LIN {X 0,Y 418.441,Z 133.979,A -85,B 0,C 180,E1 -10266.49,E2 -10266.49} C_VEL
LIN {X 0,Y 418.371,Z 133.974,A -85,B 0,C 180,E1 -10268.696,E2 -10268.696} C_VEL
LIN {X 0,Y 418.302,Z 133.992,A -85,B 0,C 180,E1 -10271.632,E2 -10271.632} C_VEL
LIN {X 0,Y 418.281,Z 134.005,A -85,B 0,C 180,E1 -10273.606,E2 -10273.606} C_VEL
LIN {X 0,Y 418.255,Z 134.002,A -85,B 0,C 180,E1 -10276.707,E2 -10276.707} C_VEL
LIN {X 0,Y 418.227,Z 134.015,A -85,B 0,C 180,E1 -10279.772,E2 -10279.772} C_VEL
LIN {X 0,Y 418.227,Z 134.007,A -85,B 0,C 180,E1 -10282.737,E2 -10282.737} C_VEL
LIN {X 0,Y 418.213,Z 134.011,A -85,B 0,C 180,E1 -10285.908,E2 -10285.908} C_VEL
LIN {X 0,Y 418.259,Z 133.991,A -85,B 0,C 180,E1 -10289.163,E2 -10289.163} C_VEL
LIN {X 0,Y 418.236,Z 134.006,A -85,B 0,C 180,E1 -10292.53,E2 -10292.53} C_VEL
LIN {X 0,Y 418.252,Z 134.011,A -85,B 0,C 180,E1 -10294.842,E2 -10294.842} C_VEL
LIN {X 0,Y 418.238,Z 133.993,A -85,B 0,C 180,E1 -10298.444,E2 -10298.444} C_VEL
LIN {X 0,Y 418.224,Z 134.012,A -85,B 0,C 180,E1 -10302.236,E2 -10302.236} C_VEL
LIN {X 0,Y 418.239,Z 133.998,A -85,B 0,C 180,E1 -10305.108,E2 -10305.108} C_VEL
LIN {X 0,Y 418.224,Z 134.008,A -85,B 0,C 180,E1 -10307.764,E2 -10307.764} C_VEL
LIN {X 0,Y 418.241,Z 134.002,A -85,B 0,C 180,E1 -10311.556,E2 -10311.556} C_VEL
LIN {X 0,Y 418.256,Z 134.008,A -85,B 0,C 180,E1 -10315.158,E2 -10315.158} C_VEL
LIN {X 0,Y 418.248,Z 134.001,A -85,B 0,C 180,E1 -10317.472,E2 -10317.472} C_VEL
LIN {X 0,Y 418.267,Z 134.005,A -85,B 0,C 180,E1 -10320.897,E2 -10320.897} C_VEL
LIN {X 0,Y 418.23,Z 134.019,A -85,B 0,C 180,E1 -10324.093,E2 -10324.093} C_VEL
LIN {X 0,Y 418.234,Z 134.012,A -85,B 0,C 180,E1 -10327.263,E2 -10327.263} C_VEL
LIN {X 0,Y 418.289,Z 134.005,A -85,B 0,C 180,E1 -10330.364,E2 -10330.364} C_VEL
LIN {X 0,Y 418.322,Z 133.996,A -85,B 0,C 180,E1 -10333.404,E2 -10333.404} C_VEL
LIN {X 0,Y 418.352,Z 133.994,A -85,B 0,C 180,E1 -10336.999,E2 -10336.999} C_VEL
LIN {X 0,Y 418.339,Z 134.079,A -85,B 0,C 180,E1 -10339.931,E2 -10339.931} C_VEL
LIN {X 0,Y 420.998,Z 145.281,A -85,B 0,C 180,E1 -10342.237,E2 -10342.237} C_VEL
LIN {X 0,Y 428.062,Z 163.126,A -85,B 0,C 180,E1 -10342.992,E2 -10342.992} C_VEL
LIN {X 0,Y 430.048,Z 172.772,A -85,B 0,C 180,E1 -10343.283,E2 -10343.283} C_VEL
LIN {X 0,Y 428.419,Z 267.206,A -85,B 0,C 180,E1 -10344.898,E2 -10344.898} C_VEL
LIN {X 0,Y 427.7,Z 273.05,A -85,B 0,C 180,E1 -10344.964,E2 -10344.964} C_VEL
LIN {X 0,Y 422.069,Z 292.069,A -85,B 0,C 180,E1 -10345.004,E2 -10345.004} C_VEL
LIN {X 0,Y 421.34,Z 297.914,A -85,B 0,C 180,E1 -10345.072,E2 -10345.072} C_VEL
LIN {X 0,Y 420.879,Z 314.557,A -85,B 0,C 180,E1 -10345.42,E2 -10345.42} C_VEL
LIN {X 0,Y 420.234,Z 329.666,A -85,B 0,C 180,E1 -10345.924,E2 -10345.924} C_VEL
LIN {X 0,Y 419.383,Z 344.848,A -85,B 0,C 180,E1 -10346.637,E2 -10346.637} C_VEL
LIN {X 0,Y 418.445,Z 358.478,A -85,B 0,C 180,E1 -10347.473,E2 -10347.473} C_VEL
LIN {X 0,Y 417.191,Z 372.593,A -85,B 0,C 180,E1 -10348.552,E2 -10348.552} C_VEL
LIN {X 0,Y 416.035,Z 385.358,A -85,B 0,C 180,E1 -10349.758,E2 -10349.758} C_VEL
LIN {X 0,Y 414.929,Z 396.123,A -85,B 0,C 180,E1 -10350.97,E2 -10350.97} C_VEL
LIN {X 0,Y 413.866,Z 407.027,A -85,B 0,C 180,E1 -10352.433,E2 -10352.433} C_VEL
LIN {X 0,Y 412.87,Z 416.307,A -85,B 0,C 180,E1 -10353.904,E2 -10353.904} C_VEL
LIN {X 0,Y 412.02,Z 425.38,A -85,B 0,C 180,E1 -10355.628,E2 -10355.628} C_VEL
LIN {X 0,Y 411.318,Z 433.108,A -85,B 0,C 180,E1 -10357.401,E2 -10357.401} C_VEL
LIN {X 0,Y 410.67,Z 440.061,A -85,B 0,C 180,E1 -10359.356,E2 -10359.356} C_VEL
LIN {X 0,Y 410.316,Z 445.653,A -85,B 0,C 180,E1 -10361.36,E2 -10361.36} C_VEL
LIN {X 0,Y 410.106,Z 448.969,A -85,B 0,C 180,E1 -10362.872,E2 -10362.872} C_VEL
LIN {X 0,Y 409.9,Z 452.257,A -85,B 0,C 180,E1 -10364.903,E2 -10364.903} C_VEL
LIN {X 0,Y 409.799,Z 454.273,A -85,B 0,C 180,E1 -10366.95,E2 -10366.95} C_VEL
LIN {X 0,Y 409.817,Z 455.04,A -85,B 0,C 180,E1 -10369.016,E2 -10369.016} C_VEL
LIN {X 0,Y 409.789,Z 454.553,A -85,B 0,C 180,E1 -10371.109,E2 -10371.109} C_VEL
LIN {X 0,Y 409.898,Z 452.759,A -85,B 0,C 180,E1 -10373.225,E2 -10373.225} C_VEL
LIN {X 0,Y 410.172,Z 449.578,A -85,B 0,C 180,E1 -10375.363,E2 -10375.363} C_VEL
LIN {X 0,Y 410.442,Z 446.011,A -85,B 0,C 180,E1 -10377.076,E2 -10377.076} C_VEL
LIN {X 0,Y 410.882,Z 440.974,A -85,B 0,C 180,E1 -10378.954,E2 -10378.954} C_VEL
LIN {X 0,Y 411.642,Z 433.496,A -85,B 0,C 180,E1 -10381.119,E2 -10381.119} C_VEL
LIN {X 0,Y 412.549,Z 425.228,A -85,B 0,C 180,E1 -10383.034,E2 -10383.034} C_VEL
LIN {X 0,Y 413.588,Z 416.553,A -85,B 0,C 180,E1 -10384.698,E2 -10384.698} C_VEL
LIN {X 0,Y 414.81,Z 406.103,A -85,B 0,C 180,E1 -10386.369,E2 -10386.369} C_VEL
LIN {X 0,Y 416.201,Z 394.576,A -85,B 0,C 180,E1 -10387.896,E2 -10387.896} C_VEL
LIN {X 0,Y 417.657,Z 381.921,A -85,B 0,C 180,E1 -10389.28,E2 -10389.28} C_VEL
LIN {X 0,Y 418.949,Z 369.71,A -85,B 0,C 180,E1 -10390.387,E2 -10390.387} C_VEL
LIN {X 0,Y 420.269,Z 355.862,A -85,B 0,C 180,E1 -10391.407,E2 -10391.407} C_VEL
LIN {X 0,Y 421.406,Z 341.436,A -85,B 0,C 180,E1 -10392.245,E2 -10392.245} C_VEL
LIN {X 0,Y 422.301,Z 326.024,A -85,B 0,C 180,E1 -10392.923,E2 -10392.923} C_VEL
LIN {X 0,Y 423.027,Z 310.672,A -85,B 0,C 180,E1 -10393.382,E2 -10393.382} C_VEL
LIN {X 0,Y 425.843,Z 173.555,A -85,B 0,C 180,E1 -10395.84,E2 -10395.84} C_VEL
LIN {X 0,Y 424.375,Z 167.927,A -85,B 0,C 180,E1 -10396.064,E2 -10396.064} C_VEL
LIN {X 0,Y 417.259,Z 152.471,A -85,B 0,C 180,E1 -10396.951,E2 -10396.951} C_VEL
LIN {X 0,Y 414.076,Z 145.825,A -85,B 0,C 180,E1 -10397.365,E2 -10397.365} C_VEL
LIN {X 0,Y 411.18,Z 134.894,A -85,B 0,C 180,E1 -10399.989,E2 -10399.989} C_VEL
LIN {X 0,Y 411.193,Z 134.893,A -85,B 0,C 180,E1 -10403.447,E2 -10403.447} C_VEL
LIN {X 0,Y 411.209,Z 134.887,A -85,B 0,C 180,E1 -10406.873,E2 -10406.873} C_VEL
LIN {X 0,Y 411.213,Z 134.883,A -85,B 0,C 180,E1 -10410.649,E2 -10410.649} C_VEL
LIN {X 0,Y 411.203,Z 134.889,A -85,B 0,C 180,E1 -10413.616,E2 -10413.616} C_VEL
LIN {X 0,Y 411.196,Z 134.882,A -85,B 0,C 180,E1 -10416.852,E2 -10416.852} C_VEL
LIN {X 0,Y 411.215,Z 134.887,A -85,B 0,C 180,E1 -10420.05,E2 -10420.05} C_VEL
LIN {X 0,Y 411.264,Z 134.879,A -85,B 0,C 180,E1 -10423.131,E2 -10423.131} C_VEL
LIN {X 0,Y 411.306,Z 134.875,A -85,B 0,C 180,E1 -10426.895,E2 -10426.895} C_VEL
LIN {X 0,Y 411.292,Z 134.875,A -85,B 0,C 180,E1 -10430.161,E2 -10430.161} C_VEL
LIN {X 0,Y 411.482,Z 134.853,A -85,B 0,C 180,E1 -10432.146,E2 -10432.146} C_VEL
LIN {X 0,Y 411.473,Z 134.849,A -85,B 0,C 180,E1 -10434.118,E2 -10434.118} C_VEL
LIN {X 0,Y 411.51,Z 134.845,A -85,B 0,C 180,E1 -10438.042,E2 -10438.042} C_VEL
LIN {X 0,Y 411.64,Z 134.833,A -85,B 0,C 180,E1 -10440,E2 -10440} C_VEL
LIN {X 0,Y 411.457,Z 134.855,A -85,B 0,C 180,E1 -10442.937,E2 -10442.937} C_VEL
LIN {X 0,Y 411.424,Z 134.861,A -85,B 0,C 180,E1 -10446.867,E2 -10446.867} C_VEL
LIN {X 0,Y 411.291,Z 134.876,A -85,B 0,C 180,E1 -10449.838,E2 -10449.838} C_VEL
LIN {X 0,Y 411.305,Z 134.873,A -85,B 0,C 180,E1 -10453.104,E2 -10453.104} C_VEL
LIN {X 0,Y 411.256,Z 134.879,A -85,B 0,C 180,E1 -10456.888,E2 -10456.888} C_VEL
LIN {X 0,Y 411.229,Z 134.878,A -85,B 0,C 180,E1 -10459.986,E2 -10459.986} C_VEL
LIN {X 0,Y 411.202,Z 134.886,A -85,B 0,C 180,E1 -10463.147,E2 -10463.147} C_VEL
LIN {X 0,Y 411.236,Z 134.881,A -85,B 0,C 180,E1 -10466.381,E2 -10466.381} C_VEL
LIN {X 0,Y 411.199,Z 134.884,A -85,B 0,C 180,E1 -10469.712,E2 -10469.712} C_VEL
LIN {X 0,Y 411.204,Z 134.888,A -85,B 0,C 180,E1 -10473.156,E2 -10473.156} C_VEL
LIN {X 0,Y 411.19,Z 134.892,A -85,B 0,C 180,E1 -10476.552,E2 -10476.552} C_VEL
LIN {X 0,Y 411.209,Z 134.88,A -85,B 0,C 180,E1 -10479.727,E2 -10479.727} C_VEL
LIN {X 0,Y 411.171,Z 134.88,A -85,B 0,C 180,E1 -10483.134,E2 -10483.134} C_VEL
LIN {X 0,Y 411.166,Z 134.891,A -85,B 0,C 180,E1 -10485.881,E2 -10485.881} C_VEL
LIN {X 0,Y 411.162,Z 134.894,A -85,B 0,C 180,E1 -10488.772,E2 -10488.772} C_VEL
LIN {X 0,Y 411.204,Z 134.89,A -85,B 0,C 180,E1 -10491.831,E2 -10491.831} C_VEL
LIN {X 0,Y 411.209,Z 134.884,A -85,B 0,C 180,E1 -10495.122,E2 -10495.122} C_VEL
LIN {X 0,Y 411.243,Z 135.042,A -85,B 0,C 180,E1 -10495.74,E2 -10495.74} C_VEL
LIN {X 0,Y 414.853,Z 148.022,A -85,B 0,C 180,E1 -10498.606,E2 -10498.606} C_VEL
LIN {X 0,Y 417.936,Z 161.061,A -85,B 0,C 180,E1 -10501.282,E2 -10501.282} C_VEL
LIN {X 0,Y 418.261,Z 164.539,A -85,B 0,C 180,E1 -10501.935,E2 -10501.935} C_VEL
LIN {X 0,Y 418.226,Z 165.397,A -85,B 0,C 180,E1 -10502.043,E2 -10502.043} C_VEL
LIN {X 0,Y 423.133,Z 187.563,A -85,B 0,C 180,E1 -10502.878,E2 -10502.878} C_VEL
LIN {X 0,Y 425.453,Z 200.436,A -85,B 0,C 180,E1 -10503.308,E2 -10503.308} C_VEL
LIN {X 0,Y 422.697,Z 331.171,A -85,B 0,C 180,E1 -10505.635,E2 -10505.635} C_VEL
LIN {X 0,Y 421.899,Z 347.287,A -85,B 0,C 180,E1 -10506.109,E2 -10506.109} C_VEL
LIN {X 0,Y 420.932,Z 361.413,A -85,B 0,C 180,E1 -10506.712,E2 -10506.712} C_VEL
LIN {X 0,Y 419.721,Z 375.189,A -85,B 0,C 180,E1 -10507.479,E2 -10507.479} C_VEL
LIN {X 0,Y 418.437,Z 388.837,A -85,B 0,C 180,E1 -10508.444,E2 -10508.444} C_VEL
LIN {X 0,Y 417.061,Z 401.409,A -85,B 0,C 180,E1 -10509.534,E2 -10509.534} C_VEL
LIN {X 0,Y 415.612,Z 414.171,A -85,B 0,C 180,E1 -10510.875,E2 -10510.875} C_VEL
LIN {X 0,Y 414.372,Z 424.885,A -85,B 0,C 180,E1 -10512.225,E2 -10512.225} C_VEL
LIN {X 0,Y 413.182,Z 434.829,A -85,B 0,C 180,E1 -10513.701,E2 -10513.701} C_VEL
LIN {X 0,Y 412.121,Z 444.59,A -85,B 0,C 180,E1 -10515.432,E2 -10515.432} C_VEL
LIN {X 0,Y 411.274,Z 452.755,A -85,B 0,C 180,E1 -10517.165,E2 -10517.165} C_VEL
LIN {X 0,Y 410.863,Z 458.598,A -85,B 0,C 180,E1 -10518.656,E2 -10518.656} C_VEL
LIN {X 0,Y 410.339,Z 465.055,A -85,B 0,C 180,E1 -10520.636,E2 -10520.636} C_VEL
LIN {X 0,Y 410.09,Z 470.101,A -85,B 0,C 180,E1 -10522.616,E2 -10522.616} C_VEL
LIN {X 0,Y 409.974,Z 473.042,A -85,B 0,C 180,E1 -10524.097,E2 -10524.097} C_VEL
LIN {X 0,Y 409.882,Z 475.851,A -85,B 0,C 180,E1 -10526.068,E2 -10526.068} C_VEL
LIN {X 0,Y 409.96,Z 477.491,A -85,B 0,C 180,E1 -10528.036,E2 -10528.036} C_VEL
LIN {X 0,Y 409.923,Z 477.989,A -85,B 0,C 180,E1 -10530,E2 -10530} C_VEL
LIN {X 0,Y 409.961,Z 477.332,A -85,B 0,C 180,E1 -10531.965,E2 -10531.965} C_VEL
LIN {X 0,Y 409.886,Z 475.46,A -85,B 0,C 180,E1 -10533.933,E2 -10533.933} C_VEL
LIN {X 0,Y 409.987,Z 472.398,A -85,B 0,C 180,E1 -10535.904,E2 -10535.904} C_VEL
LIN {X 0,Y 410.139,Z 468.066,A -85,B 0,C 180,E1 -10537.88,E2 -10537.88} C_VEL
LIN {X 0,Y 410.356,Z 462.344,A -85,B 0,C 180,E1 -10539.862,E2 -10539.862} C_VEL
LIN {X 0,Y 410.885,Z 455.084,A -85,B 0,C 180,E1 -10541.845,E2 -10541.845} C_VEL
LIN {X 0,Y 411.481,Z 447.245,A -85,B 0,C 180,E1 -10543.595,E2 -10543.595} C_VEL
LIN {X 0,Y 412.329,Z 437.934,A -85,B 0,C 180,E1 -10545.319,E2 -10545.319} C_VEL
LIN {X 0,Y 413.323,Z 428.406,A -85,B 0,C 180,E1 -10546.802,E2 -10546.802} C_VEL
LIN {X 0,Y 414.427,Z 417.293,A -85,B 0,C 180,E1 -10548.256,E2 -10548.256} C_VEL
LIN {X 0,Y 415.66,Z 404.612,A -85,B 0,C 180,E1 -10549.637,E2 -10549.637} C_VEL
LIN {X 0,Y 416.96,Z 390.852,A -85,B 0,C 180,E1 -10550.859,E2 -10550.859} C_VEL
LIN {X 0,Y 418.133,Z 377.332,A -85,B 0,C 180,E1 -10551.832,E2 -10551.832} C_VEL
LIN {X 0,Y 419.24,Z 362.385,A -85,B 0,C 180,E1 -10552.679,E2 -10552.679} C_VEL
LIN {X 0,Y 420.108,Z 347.502,A -85,B 0,C 180,E1 -10553.313,E2 -10553.313} C_VEL
LIN {X 0,Y 420.82,Z 332.224,A -85,B 0,C 180,E1 -10553.76,E2 -10553.76} C_VEL
LIN {X 0,Y 423.17,Z 199.963,A -85,B 0,C 180,E1 -10556.077,E2 -10556.077} C_VEL
LIN {X 0,Y 416.874,Z 165.615,A -85,B 0,C 180,E1 -10557.112,E2 -10557.112} C_VEL
LIN {X 0,Y 417.205,Z 161.049,A -85,B 0,C 180,E1 -10557.87,E2 -10557.87} C_VEL
LIN {X 0,Y 415.303,Z 151.738,A -85,B 0,C 180,E1 -10559.594,E2 -10559.594} C_VEL
LIN {X 0,Y 411.601,Z 136.533,A -85,B 0,C 180,E1 -10562.538,E2 -10562.538} C_VEL
LIN {X 0,Y 411.225,Z 134.89,A -85,B 0,C 180,E1 -10562.907,E2 -10562.907} C_VEL
LIN {X 0,Y 411.2,Z 134.895,A -85,B 0,C 180,E1 -10565.529,E2 -10565.529} C_VEL
LIN {X 0,Y 411.212,Z 134.888,A -85,B 0,C 180,E1 -10569.226,E2 -10569.226} C_VEL
LIN {X 0,Y 411.179,Z 134.89,A -85,B 0,C 180,E1 -10572.696,E2 -10572.696} C_VEL
LIN {X 0,Y 411.17,Z 134.897,A -85,B 0,C 180,E1 -10575.882,E2 -10575.882} C_VEL
LIN {X 0,Y 411.165,Z 134.894,A -85,B 0,C 180,E1 -10578.772,E2 -10578.772} C_VEL
LIN {X 0,Y 411.192,Z 134.888,A -85,B 0,C 180,E1 -10582.026,E2 -10582.026} C_VEL
LIN {X 0,Y 411.207,Z 134.888,A -85,B 0,C 180,E1 -10585.667,E2 -10585.667} C_VEL
LIN {X 0,Y 411.192,Z 134.892,A -85,B 0,C 180,E1 -10589.153,E2 -10589.153} C_VEL
LIN {X 0,Y 411.181,Z 134.876,A -85,B 0,C 180,E1 -10591.407,E2 -10591.407} C_VEL
LIN {X 0,Y 411.23,Z 134.882,A -85,B 0,C 180,E1 -10594.93,E2 -10594.93} C_VEL
LIN {X 0,Y 411.209,Z 134.881,A -85,B 0,C 180,E1 -10597.914,E2 -10597.914} C_VEL
LIN {X 0,Y 411.223,Z 134.886,A -85,B 0,C 180,E1 -10601.052,E2 -10601.052} C_VEL
LIN {X 0,Y 411.257,Z 134.877,A -85,B 0,C 180,E1 -10604.132,E2 -10604.132} C_VEL
LIN {X 0,Y 411.308,Z 134.87,A -85,B 0,C 180,E1 -10607.166,E2 -10607.166} C_VEL
LIN {X 0,Y 411.294,Z 134.877,A -85,B 0,C 180,E1 -10610.162,E2 -10610.162} C_VEL
LIN {X 0,Y 411.395,Z 134.86,A -85,B 0,C 180,E1 -10613.132,E2 -10613.132} C_VEL
LIN {X 0,Y 411.293,Z 134.874,A -85,B 0,C 180,E1 -10615.099,E2 -10615.099} C_VEL
LIN {X 0,Y 411.507,Z 134.838,A -85,B 0,C 180,E1 -10618.043,E2 -10618.043} C_VEL
LIN {X 0,Y 411.382,Z 134.852,A -85,B 0,C 180,E1 -10620.979,E2 -10620.979} C_VEL
LIN {X 0,Y 411.43,Z 134.855,A -85,B 0,C 180,E1 -10622.938,E2 -10622.938} C_VEL
LIN {X 0,Y 411.395,Z 134.855,A -85,B 0,C 180,E1 -10626.868,E2 -10626.868} C_VEL
LIN {X 0,Y 411.278,Z 134.857,A -85,B 0,C 180,E1 -10629.84,E2 -10629.84} C_VEL
LIN {X 0,Y 411.305,Z 134.87,A -85,B 0,C 180,E1 -10633.1,E2 -10633.1} C_VEL
LIN {X 0,Y 411.209,Z 134.88,A -85,B 0,C 180,E1 -10636.891,E2 -10636.891} C_VEL
LIN {X 0,Y 411.181,Z 134.89,A -85,B 0,C 180,E1 -10639.99,E2 -10639.99} C_VEL
LIN {X 0,Y 411.187,Z 134.887,A -85,B 0,C 180,E1 -10643.149,E2 -10643.149} C_VEL
LIN {X 0,Y 411.168,Z 134.887,A -85,B 0,C 180,E1 -10646.386,E2 -10646.386} C_VEL
LIN {X 0,Y 411.197,Z 134.87,A -85,B 0,C 180,E1 -10649.714,E2 -10649.714} C_VEL
LIN {X 0,Y 411.207,Z 134.888,A -85,B 0,C 180,E1 -10653.156,E2 -10653.156} C_VEL
LIN {X 0,Y 411.193,Z 134.884,A -85,B 0,C 180,E1 -10656.551,E2 -10656.551} C_VEL
LIN {X 0,Y 411.172,Z 134.883,A -85,B 0,C 180,E1 -10659.72,E2 -10659.72} C_VEL
LIN {X 0,Y 411.167,Z 134.891,A -85,B 0,C 180,E1 -10663.135,E2 -10663.135} C_VEL
LIN {X 0,Y 411.168,Z 134.875,A -85,B 0,C 180,E1 -10665.882,E2 -10665.882} C_VEL
LIN {X 0,Y 411.153,Z 134.898,A -85,B 0,C 180,E1 -10668.774,E2 -10668.774} C_VEL
LIN {X 0,Y 411.189,Z 134.882,A -85,B 0,C 180,E1 -10672.025,E2 -10672.025} C_VEL
LIN {X 0,Y 411.208,Z 134.886,A -85,B 0,C 180,E1 -10675.123,E2 -10675.123} C_VEL
LIN {X 0,Y 411.17,Z 134.885,A -85,B 0,C 180,E1 -10678.002,E2 -10678.002} C_VEL
LIN {X 0,Y 411.181,Z 134.887,A -85,B 0,C 180,E1 -10681.407,E2 -10681.407} C_VEL
LIN {X 0,Y 411.217,Z 134.887,A -85,B 0,C 180,E1 -10684.934,E2 -10684.934} C_VEL
LIN {X 0,Y 411.209,Z 134.891,A -85,B 0,C 180,E1 -10687.913,E2 -10687.913} C_VEL
LIN {X 0,Y 411.224,Z 134.882,A -85,B 0,C 180,E1 -10691.051,E2 -10691.051} C_VEL
LIN {X 0,Y 411.259,Z 134.885,A -85,B 0,C 180,E1 -10694.131,E2 -10694.131} C_VEL
LIN {X 0,Y 411.309,Z 134.873,A -85,B 0,C 180,E1 -10697.165,E2 -10697.165} C_VEL
LIN {X 0,Y 411.325,Z 135.028,A -85,B 0,C 180,E1 -10699.602,E2 -10699.602} C_VEL
LIN {X 0,Y 413.748,Z 145.214,A -85,B 0,C 180,E1 -10701.78,E2 -10701.78} C_VEL
LIN {X 0,Y 421.775,Z 165.181,A -85,B 0,C 180,E1 -10702.655,E2 -10702.655} C_VEL
LIN {X 0,Y 423.524,Z 173.691,A -85,B 0,C 180,E1 -10702.917,E2 -10702.917} C_VEL
LIN {X 0,Y 421.34,Z 297.914,A -85,B 0,C 180,E1 -10705.072,E2 -10705.072} C_VEL
LIN {X 0,Y 420.592,Z 303.752,A -85,B 0,C 180,E1 -10705.142,E2 -10705.142} C_VEL
LIN {X 0,Y 415.162,Z 320.706,A -85,B 0,C 180,E1 -10705.306,E2 -10705.306} C_VEL
LIN {X 0,Y 413.9,Z 326.428,A -85,B 0,C 180,E1 -10705.451,E2 -10705.451} C_VEL
LIN {X 0,Y 413.703,Z 328.271,A -85,B 0,C 180,E1 -10705.52,E2 -10705.52} C_VEL
LIN {X 0,Y 412.892,Z 342.301,A -85,B 0,C 180,E1 -10706.157,E2 -10706.157} C_VEL
LIN {X 0,Y 411.936,Z 355.69,A -85,B 0,C 180,E1 -10706.943,E2 -10706.943} C_VEL
LIN {X 0,Y 410.815,Z 368.911,A -85,B 0,C 180,E1 -10707.916,E2 -10707.916} C_VEL
LIN {X 0,Y 409.486,Z 382.428,A -85,B 0,C 180,E1 -10709.139,E2 -10709.139} C_VEL
LIN {X 0,Y 408.33,Z 394.346,A -85,B 0,C 180,E1 -10710.457,E2 -10710.457} C_VEL
LIN {X 0,Y 407.077,Z 405.842,A -85,B 0,C 180,E1 -10711.978,E2 -10711.978} C_VEL
LIN {X 0,Y 405.912,Z 416.74,A -85,B 0,C 180,E1 -10713.722,E2 -10713.722} C_VEL
LIN {X 0,Y 405.008,Z 425.784,A -85,B 0,C 180,E1 -10715.476,E2 -10715.476} C_VEL
LIN {X 0,Y 404.238,Z 433.991,A -85,B 0,C 180,E1 -10717.409,E2 -10717.409} C_VEL
LIN {X 0,Y 403.709,Z 439.572,A -85,B 0,C 180,E1 -10719.014,E2 -10719.014} C_VEL
LIN {X 0,Y 403.288,Z 445.322,A -85,B 0,C 180,E1 -10721.051,E2 -10721.051} C_VEL
LIN {X 0,Y 402.967,Z 449.703,A -85,B 0,C 180,E1 -10723.104,E2 -10723.104} C_VEL
LIN {X 0,Y 402.792,Z 452.796,A -85,B 0,C 180,E1 -10725.172,E2 -10725.172} C_VEL
LIN {X 0,Y 402.681,Z 454.652,A -85,B 0,C 180,E1 -10727.259,E2 -10727.259} C_VEL
LIN {X 0,Y 402.734,Z 455.268,A -85,B 0,C 180,E1 -10729.363,E2 -10729.363} C_VEL
LIN {X 0,Y 402.712,Z 454.606,A -85,B 0,C 180,E1 -10731.499,E2 -10731.499} C_VEL
LIN {X 0,Y 402.837,Z 452.611,A -85,B 0,C 180,E1 -10733.657,E2 -10733.657} C_VEL
LIN {X 0,Y 403.184,Z 449.215,A -85,B 0,C 180,E1 -10735.835,E2 -10735.835} C_VEL
LIN {X 0,Y 403.567,Z 444.289,A -85,B 0,C 180,E1 -10738.047,E2 -10738.047} C_VEL
LIN {X 0,Y 404.107,Z 438.965,A -85,B 0,C 180,E1 -10739.869,E2 -10739.869} C_VEL
LIN {X 0,Y 404.844,Z 432.329,A -85,B 0,C 180,E1 -10741.719,E2 -10741.719} C_VEL
LIN {X 0,Y 405.834,Z 423.839,A -85,B 0,C 180,E1 -10743.652,E2 -10743.652} C_VEL
LIN {X 0,Y 407.037,Z 414.852,A -85,B 0,C 180,E1 -10745.339,E2 -10745.339} C_VEL
LIN {X 0,Y 408.367,Z 404.007,A -85,B 0,C 180,E1 -10747.038,E2 -10747.038} C_VEL
LIN {X 0,Y 409.881,Z 392.013,A -85,B 0,C 180,E1 -10748.587,E2 -10748.587} C_VEL
LIN {X 0,Y 411.295,Z 380.226,A -85,B 0,C 180,E1 -10749.85,E2 -10749.85} C_VEL
LIN {X 0,Y 412.65,Z 367.609,A -85,B 0,C 180,E1 -10750.973,E2 -10750.973} C_VEL
LIN {X 0,Y 414.027,Z 353.805,A -85,B 0,C 180,E1 -10751.966,E2 -10751.966} C_VEL
LIN {X 0,Y 415.106,Z 339.984,A -85,B 0,C 180,E1 -10752.758,E2 -10752.758} C_VEL
LIN {X 0,Y 416.078,Z 325.123,A -85,B 0,C 180,E1 -10753.397,E2 -10753.397} C_VEL
LIN {X 0,Y 416.755,Z 310.055,A -85,B 0,C 180,E1 -10753.846,E2 -10753.846} C_VEL
LIN {X 0,Y 419.788,Z 175.648,A -85,B 0,C 180,E1 -10756.278,E2 -10756.278} C_VEL
LIN {X 0,Y 418.63,Z 170.913,A -85,B 0,C 180,E1 -10756.467,E2 -10756.467} C_VEL
LIN {X 0,Y 411.223,Z 154.861,A -85,B 0,C 180,E1 -10757.415,E2 -10757.415} C_VEL
LIN {X 0,Y 406.905,Z 146.042,A -85,B 0,C 180,E1 -10757.996,E2 -10757.996} C_VEL
LIN {X 0,Y 404.161,Z 135.769,A -85,B 0,C 180,E1 -10760.561,E2 -10760.561} C_VEL
LIN {X 0,Y 404.142,Z 135.773,A -85,B 0,C 180,E1 -10763.753,E2 -10763.753} C_VEL
LIN {X 0,Y 404.172,Z 135.766,A -85,B 0,C 180,E1 -10766.579,E2 -10766.579} C_VEL
LIN {X 0,Y 404.145,Z 135.769,A -85,B 0,C 180,E1 -10769.714,E2 -10769.714} C_VEL
LIN {X 0,Y 404.152,Z 135.765,A -85,B 0,C 180,E1 -10773.119,E2 -10773.119} C_VEL
LIN {X 0,Y 404.16,Z 135.754,A -85,B 0,C 180,E1 -10776.424,E2 -10776.424} C_VEL
LIN {X 0,Y 404.192,Z 135.761,A -85,B 0,C 180,E1 -10779.874,E2 -10779.874} C_VEL
LIN {X 0,Y 404.216,Z 135.756,A -85,B 0,C 180,E1 -10782.993,E2 -10782.993} C_VEL
LIN {X 0,Y 404.283,Z 135.75,A -85,B 0,C 180,E1 -10786.938,E2 -10786.938} C_VEL
LIN {X 0,Y 404.258,Z 135.753,A -85,B 0,C 180,E1 -10789.988,E2 -10789.988} C_VEL
LIN {X 0,Y 404.41,Z 135.735,A -85,B 0,C 180,E1 -10793.012,E2 -10793.012} C_VEL
LIN {X 0,Y 404.28,Z 135.745,A -85,B 0,C 180,E1 -10795.013,E2 -10795.013} C_VEL
LIN {X 0,Y 404.479,Z 135.72,A -85,B 0,C 180,E1 -10798.008,E2 -10798.008} C_VEL
LIN {X 0,Y 404.61,Z 135.709,A -85,B 0,C 180,E1 -10800,E2 -10800} C_VEL
LIN {X 0,Y 404.415,Z 135.733,A -85,B 0,C 180,E1 -10802.988,E2 -10802.988} C_VEL
LIN {X 0,Y 404.37,Z 135.741,A -85,B 0,C 180,E1 -10806.988,E2 -10806.988} C_VEL
LIN {X 0,Y 404.256,Z 135.751,A -85,B 0,C 180,E1 -10810.011,E2 -10810.011} C_VEL
LIN {X 0,Y 404.266,Z 135.75,A -85,B 0,C 180,E1 -10813.211,E2 -10813.211} C_VEL
LIN {X 0,Y 404.215,Z 135.757,A -85,B 0,C 180,E1 -10817.007,E2 -10817.007} C_VEL
LIN {X 0,Y 404.163,Z 135.76,A -85,B 0,C 180,E1 -10820.351,E2 -10820.351} C_VEL
LIN {X 0,Y 404.168,Z 135.762,A -85,B 0,C 180,E1 -10823.574,E2 -10823.574} C_VEL
LIN {X 0,Y 404.182,Z 135.759,A -85,B 0,C 180,E1 -10825.766,E2 -10825.766} C_VEL
LIN {X 0,Y 404.194,Z 135.761,A -85,B 0,C 180,E1 -10827.999,E2 -10827.999} C_VEL
LIN {X 0,Y 404.137,Z 135.766,A -85,B 0,C 180,E1 -10831.558,E2 -10831.558} C_VEL
LIN {X 0,Y 404.182,Z 135.761,A -85,B 0,C 180,E1 -10835.016,E2 -10835.016} C_VEL
LIN {X 0,Y 404.15,Z 135.753,A -85,B 0,C 180,E1 -10838.757,E2 -10838.757} C_VEL
LIN {X 0,Y 404.121,Z 135.771,A -85,B 0,C 180,E1 -10841.6,E2 -10841.6} C_VEL
LIN {X 0,Y 404.143,Z 135.768,A -85,B 0,C 180,E1 -10844.522,E2 -10844.522} C_VEL
LIN {X 0,Y 404.135,Z 135.761,A -85,B 0,C 180,E1 -10847.296,E2 -10847.296} C_VEL
LIN {X 0,Y 404.167,Z 135.759,A -85,B 0,C 180,E1 -10849.955,E2 -10849.955} C_VEL
LIN {X 0,Y 404.135,Z 135.765,A -85,B 0,C 180,E1 -10853.125,E2 -10853.125} C_VEL
LIN {X 0,Y 404.209,Z 135.912,A -85,B 0,C 180,E1 -10855.177,E2 -10855.177} C_VEL
LIN {X 0,Y 408.054,Z 149.82,A -85,B 0,C 180,E1 -10858.329,E2 -10858.329} C_VEL
LIN {X 0,Y 410.845,Z 161.232,A -85,B 0,C 180,E1 -10860.74,E2 -10860.74} C_VEL
LIN {X 0,Y 411.602,Z 165.033,A -85,B 0,C 180,E1 -10861.481,E2 -10861.481} C_VEL
LIN {X 0,Y 416.366,Z 185.416,A -85,B 0,C 180,E1 -10862.293,E2 -10862.293} C_VEL
LIN {X 0,Y 419.249,Z 201.665,A -85,B 0,C 180,E1 -10862.85,E2 -10862.85} C_VEL
LIN {X 0,Y 416.375,Z 331.674,A -85,B 0,C 180,E1 -10865.208,E2 -10865.208} C_VEL
LIN {X 0,Y 415.524,Z 347.469,A -85,B 0,C 180,E1 -10865.686,E2 -10865.686} C_VEL
LIN {X 0,Y 414.567,Z 360.89,A -85,B 0,C 180,E1 -10866.268,E2 -10866.268} C_VEL
LIN {X 0,Y 413.194,Z 375.692,A -85,B 0,C 180,E1 -10867.103,E2 -10867.103} C_VEL
LIN {X 0,Y 411.686,Z 390.751,A -85,B 0,C 180,E1 -10868.205,E2 -10868.205} C_VEL
LIN {X 0,Y 410.279,Z 402.95,A -85,B 0,C 180,E1 -10869.311,E2 -10869.311} C_VEL
LIN {X 0,Y 408.743,Z 415.416,A -85,B 0,C 180,E1 -10870.672,E2 -10870.672} C_VEL
LIN {X 0,Y 407.374,Z 426.78,A -85,B 0,C 180,E1 -10872.169,E2 -10872.169} C_VEL
LIN {X 0,Y 406.157,Z 436.373,A -85,B 0,C 180,E1 -10873.669,E2 -10873.669} C_VEL
LIN {X 0,Y 405.045,Z 445.823,A -85,B 0,C 180,E1 -10875.429,E2 -10875.429} C_VEL
LIN {X 0,Y 404.205,Z 453.718,A -85,B 0,C 180,E1 -10877.192,E2 -10877.192} C_VEL
LIN {X 0,Y 403.672,Z 460.307,A -85,B 0,C 180,E1 -10878.959,E2 -10878.959} C_VEL
LIN {X 0,Y 403.196,Z 466.38,A -85,B 0,C 180,E1 -10880.975,E2 -10880.975} C_VEL
LIN {X 0,Y 402.973,Z 471.059,A -85,B 0,C 180,E1 -10882.988,E2 -10882.988} C_VEL
LIN {X 0,Y 402.851,Z 474.451,A -85,B 0,C 180,E1 -10884.996,E2 -10884.996} C_VEL
LIN {X 0,Y 402.799,Z 476.644,A -85,B 0,C 180,E1 -10887,E2 -10887} C_VEL
LIN {X 0,Y 402.859,Z 477.688,A -85,B 0,C 180,E1 -10889.001,E2 -10889.001} C_VEL
LIN {X 0,Y 402.859,Z 477.594,A -85,B 0,C 180,E1 -10891,E2 -10891} C_VEL
LIN {X 0,Y 402.803,Z 476.311,A -85,B 0,C 180,E1 -10893.001,E2 -10893.001} C_VEL
LIN {X 0,Y 402.87,Z 473.826,A -85,B 0,C 180,E1 -10895.004,E2 -10895.004} C_VEL
LIN {X 0,Y 402.983,Z 470.113,A -85,B 0,C 180,E1 -10897.013,E2 -10897.013} C_VEL
LIN {X 0,Y 403.155,Z 465.072,A -85,B 0,C 180,E1 -10899.027,E2 -10899.027} C_VEL
LIN {X 0,Y 403.593,Z 458.574,A -85,B 0,C 180,E1 -10901.044,E2 -10901.044} C_VEL
LIN {X 0,Y 404.117,Z 451.558,A -85,B 0,C 180,E1 -10902.811,E2 -10902.811} C_VEL
LIN {X 0,Y 404.866,Z 443.102,A -85,B 0,C 180,E1 -10904.579,E2 -10904.579} C_VEL
LIN {X 0,Y 405.882,Z 432.899,A -85,B 0,C 180,E1 -10906.343,E2 -10906.343} C_VEL
LIN {X 0,Y 406.999,Z 422.476,A -85,B 0,C 180,E1 -10907.849,E2 -10907.849} C_VEL
LIN {X 0,Y 408.253,Z 409.962,A -85,B 0,C 180,E1 -10909.353,E2 -10909.353} C_VEL
LIN {X 0,Y 409.548,Z 397.407,A -85,B 0,C 180,E1 -10910.597,E2 -10910.597} C_VEL
LIN {X 0,Y 410.815,Z 383.632,A -85,B 0,C 180,E1 -10911.713,E2 -10911.713} C_VEL
LIN {X 0,Y 412.038,Z 369.622,A -85,B 0,C 180,E1 -10912.618,E2 -10912.618} C_VEL
LIN {X 0,Y 413.024,Z 355.326,A -85,B 0,C 180,E1 -10913.338,E2 -10913.338} C_VEL
LIN {X 0,Y 413.857,Z 339.847,A -85,B 0,C 180,E1 -10913.906,E2 -10913.906} C_VEL
LIN {X 0,Y 414.382,Z 323.621,A -85,B 0,C 180,E1 -10914.286,E2 -10914.286} C_VEL
LIN {X 0,Y 416.647,Z 200.722,A -85,B 0,C 180,E1 -10916.448,E2 -10916.448} C_VEL
LIN {X 0,Y 410.095,Z 165.475,A -85,B 0,C 180,E1 -10917.528,E2 -10917.528} C_VEL
LIN {X 0,Y 410.328,Z 162.1,A -85,B 0,C 180,E1 -10918.101,E2 -10918.101} C_VEL
LIN {X 0,Y 407.256,Z 148.332,A -85,B 0,C 180,E1 -10920.727,E2 -10920.727} C_VEL
LIN {X 0,Y 404.18,Z 135.769,A -85,B 0,C 180,E1 -10923.24,E2 -10923.24} C_VEL
LIN {X 0,Y 404.145,Z 135.771,A -85,B 0,C 180,E1 -10926.247,E2 -10926.247} C_VEL
LIN {X 0,Y 404.153,Z 135.766,A -85,B 0,C 180,E1 -10928.758,E2 -10928.758} C_VEL
LIN {X 0,Y 404.12,Z 135.773,A -85,B 0,C 180,E1 -10931.6,E2 -10931.6} C_VEL
LIN {X 0,Y 404.147,Z 135.769,A -85,B 0,C 180,E1 -10934.523,E2 -10934.523} C_VEL
LIN {X 0,Y 404.138,Z 135.774,A -85,B 0,C 180,E1 -10937.296,E2 -10937.296} C_VEL
LIN {X 0,Y 404.171,Z 135.761,A -85,B 0,C 180,E1 -10939.956,E2 -10939.956} C_VEL
LIN {X 0,Y 404.138,Z 135.77,A -85,B 0,C 180,E1 -10943.126,E2 -10943.126} C_VEL
LIN {X 0,Y 404.147,Z 135.765,A -85,B 0,C 180,E1 -10946.188,E2 -10946.188} C_VEL
LIN {X 0,Y 404.147,Z 135.764,A -85,B 0,C 180,E1 -10949.715,E2 -10949.715} C_VEL
LIN {X 0,Y 404.127,Z 135.754,A -85,B 0,C 180,E1 -10953.118,E2 -10953.118} C_VEL
LIN {X 0,Y 404.169,Z 135.763,A -85,B 0,C 180,E1 -10956.426,E2 -10956.426} C_VEL
LIN {X 0,Y 404.195,Z 135.758,A -85,B 0,C 180,E1 -10959.875,E2 -10959.875} C_VEL
LIN {X 0,Y 404.22,Z 135.754,A -85,B 0,C 180,E1 -10962.994,E2 -10962.994} C_VEL
LIN {X 0,Y 404.287,Z 135.746,A -85,B 0,C 180,E1 -10966.939,E2 -10966.939} C_VEL
LIN {X 0,Y 404.26,Z 135.752,A -85,B 0,C 180,E1 -10969.989,E2 -10969.989} C_VEL
LIN {X 0,Y 404.345,Z 135.739,A -85,B 0,C 180,E1 -10973.012,E2 -10973.012} C_VEL
LIN {X 0,Y 404.265,Z 135.75,A -85,B 0,C 180,E1 -10975.014,E2 -10975.014} C_VEL
LIN {X 0,Y 404.476,Z 135.713,A -85,B 0,C 180,E1 -10978.009,E2 -10978.009} C_VEL
LIN {X 0,Y 404.352,Z 135.727,A -85,B 0,C 180,E1 -10980.996,E2 -10980.996} C_VEL
LIN {X 0,Y 404.364,Z 135.735,A -85,B 0,C 180,E1 -10982.989,E2 -10982.989} C_VEL
LIN {X 0,Y 404.343,Z 135.735,A -85,B 0,C 180,E1 -10986.484,E2 -10986.484} C_VEL
LIN {X 0,Y 404.259,Z 135.73,A -85,B 0,C 180,E1 -10989.002,E2 -10989.002} C_VEL
LIN {X 0,Y 404.248,Z 135.748,A -85,B 0,C 180,E1 -10992.042,E2 -10992.042} C_VEL
LIN {X 0,Y 404.161,Z 135.763,A -85,B 0,C 180,E1 -10995.12,E2 -10995.12} C_VEL
LIN {X 0,Y 404.122,Z 135.768,A -85,B 0,C 180,E1 -10998.243,E2 -10998.243} C_VEL
LIN {X 0,Y 404.128,Z 135.768,A -85,B 0,C 180,E1 -11001.42,E2 -11001.42} C_VEL
LIN {X 0,Y 404.138,Z 135.766,A -85,B 0,C 180,E1 -11004.669,E2 -11004.669} C_VEL
LIN {X 0,Y 404.104,Z 135.757,A -85,B 0,C 180,E1 -11008.007,E2 -11008.007} C_VEL
LIN {X 0,Y 404.144,Z 135.749,A -85,B 0,C 180,E1 -11010.286,E2 -11010.286} C_VEL
LIN {X 0,Y 404.141,Z 135.766,A -85,B 0,C 180,E1 -11013.813,E2 -11013.813} C_VEL
LIN {X 0,Y 404.135,Z 135.757,A -85,B 0,C 180,E1 -11016.874,E2 -11016.874} C_VEL
LIN {X 0,Y 404.122,Z 135.761,A -85,B 0,C 180,E1 -11020.075,E2 -11020.075} C_VEL
LIN {X 0,Y 404.147,Z 135.766,A -85,B 0,C 180,E1 -11023.082,E2 -11023.082} C_VEL
LIN {X 0,Y 404.125,Z 135.752,A -85,B 0,C 180,E1 -11025.922,E2 -11025.922} C_VEL
LIN {X 0,Y 404.107,Z 135.773,A -85,B 0,C 180,E1 -11028.633,E2 -11028.633} C_VEL
LIN {X 0,Y 404.144,Z 135.758,A -85,B 0,C 180,E1 -11031.495,E2 -11031.495} C_VEL
LIN {X 0,Y 404.183,Z 135.762,A -85,B 0,C 180,E1 -11034.983,E2 -11034.983} C_VEL
LIN {X 0,Y 404.144,Z 135.766,A -85,B 0,C 180,E1 -11038.442,E2 -11038.442} C_VEL
LIN {X 0,Y 404.157,Z 135.763,A -85,B 0,C 180,E1 -11040.862,E2 -11040.862} C_VEL
LIN {X 0,Y 404.142,Z 135.773,A -85,B 0,C 180,E1 -11044.23,E2 -11044.23} C_VEL
LIN {X 0,Y 404.172,Z 135.765,A -85,B 0,C 180,E1 -11047.508,E2 -11047.508} C_VEL
LIN {X 0,Y 404.168,Z 135.761,A -85,B 0,C 180,E1 -11050.707,E2 -11050.707} C_VEL
LIN {X 0,Y 404.226,Z 135.756,A -85,B 0,C 180,E1 -11053.848,E2 -11053.848} C_VEL
LIN {X 0,Y 404.288,Z 135.744,A -85,B 0,C 180,E1 -11056.939,E2 -11056.939} C_VEL
LIN {X 0,Y 404.267,Z 135.832,A -85,B 0,C 180,E1 -11059.229,E2 -11059.229} C_VEL
LIN {X 0,Y 406.547,Z 145.476,A -85,B 0,C 180,E1 -11061.324,E2 -11061.324} C_VEL
LIN {X 0,Y 415.609,Z 167.873,A -85,B 0,C 180,E1 -11062.329,E2 -11062.329} C_VEL
LIN {X 0,Y 417.02,Z 174.595,A -85,B 0,C 180,E1 -11062.542,E2 -11062.542} C_VEL
LIN {X 0,Y 414.474,Z 310.206,A -85,B 0,C 180,E1 -11064.953,E2 -11064.953} C_VEL
LIN {X 0,Y 413.86,Z 325.287,A -85,B 0,C 180,E1 -11065.403,E2 -11065.403} C_VEL
LIN {X 0,Y 413.703,Z 328.271,A -85,B 0,C 180,E1 -11065.52,E2 -11065.52} C_VEL
LIN {X 0,Y 412.154,Z 335.781,A -85,B 0,C 180,E1 -11065.778,E2 -11065.778} C_VEL
LIN {X 0,Y 406.702,Z 350.22,A -85,B 0,C 180,E1 -11066.301,E2 -11066.301} C_VEL
LIN {X 0,Y 405.351,Z 355.583,A -85,B 0,C 180,E1 -11066.595,E2 -11066.595} C_VEL
LIN {X 0,Y 405.143,Z 357.325,A -85,B 0,C 180,E1 -11066.714,E2 -11066.714} C_VEL
LIN {X 0,Y 403.883,Z 370.939,A -85,B 0,C 180,E1 -11067.756,E2 -11067.756} C_VEL
LIN {X 0,Y 402.535,Z 384.112,A -85,B 0,C 180,E1 -11068.999,E2 -11068.999} C_VEL
LIN {X 0,Y 401.242,Z 396.469,A -85,B 0,C 180,E1 -11070.422,E2 -11070.422} C_VEL
LIN {X 0,Y 400.024,Z 407.904,A -85,B 0,C 180,E1 -11072.013,E2 -11072.013} C_VEL
LIN {X 0,Y 398.806,Z 418.486,A -85,B 0,C 180,E1 -11073.789,E2 -11073.789} C_VEL
LIN {X 0,Y 397.879,Z 427.293,A -85,B 0,C 180,E1 -11075.575,E2 -11075.575} C_VEL
LIN {X 0,Y 397.26,Z 433.67,A -85,B 0,C 180,E1 -11077.113,E2 -11077.113} C_VEL
LIN {X 0,Y 396.573,Z 440.721,A -85,B 0,C 180,E1 -11079.177,E2 -11079.177} C_VEL
LIN {X 0,Y 396.176,Z 446.257,A -85,B 0,C 180,E1 -11081.252,E2 -11081.252} C_VEL
LIN {X 0,Y 395.844,Z 450.437,A -85,B 0,C 180,E1 -11083.344,E2 -11083.344} C_VEL
LIN {X 0,Y 395.68,Z 453.336,A -85,B 0,C 180,E1 -11085.451,E2 -11085.451} C_VEL
LIN {X 0,Y 395.586,Z 454.999,A -85,B 0,C 180,E1 -11087.579,E2 -11087.579} C_VEL
LIN {X 0,Y 395.622,Z 455.422,A -85,B 0,C 180,E1 -11089.726,E2 -11089.726} C_VEL
LIN {X 0,Y 395.654,Z 454.574,A -85,B 0,C 180,E1 -11091.902,E2 -11091.902} C_VEL
LIN {X 0,Y 395.792,Z 452.393,A -85,B 0,C 180,E1 -11094.104,E2 -11094.104} C_VEL
LIN {X 0,Y 396.202,Z 448.791,A -85,B 0,C 180,E1 -11096.325,E2 -11096.325} C_VEL
LIN {X 0,Y 396.633,Z 443.617,A -85,B 0,C 180,E1 -11098.582,E2 -11098.582} C_VEL
LIN {X 0,Y 397.203,Z 438.587,A -85,B 0,C 180,E1 -11100.298,E2 -11100.298} C_VEL
LIN {X 0,Y 397.937,Z 432.371,A -85,B 0,C 180,E1 -11102.033,E2 -11102.033} C_VEL
LIN {X 0,Y 399.052,Z 423.654,A -85,B 0,C 180,E1 -11104.038,E2 -11104.038} C_VEL
LIN {X 0,Y 400.451,Z 413.706,A -85,B 0,C 180,E1 -11105.905,E2 -11105.905} C_VEL
LIN {X 0,Y 401.695,Z 403.894,A -85,B 0,C 180,E1 -11107.443,E2 -11107.443} C_VEL
LIN {X 0,Y 403.34,Z 391.88,A -85,B 0,C 180,E1 -11109.01,E2 -11109.01} C_VEL
LIN {X 0,Y 404.764,Z 380.399,A -85,B 0,C 180,E1 -11110.258,E2 -11110.258} C_VEL
LIN {X 0,Y 406.221,Z 367.569,A -85,B 0,C 180,E1 -11111.415,E2 -11111.415} C_VEL
LIN {X 0,Y 407.676,Z 353.818,A -85,B 0,C 180,E1 -11112.414,E2 -11112.414} C_VEL
LIN {X 0,Y 408.765,Z 340.367,A -85,B 0,C 180,E1 -11113.196,E2 -11113.196} C_VEL
LIN {X 0,Y 409.788,Z 325.046,A -85,B 0,C 180,E1 -11113.863,E2 -11113.863} C_VEL
LIN {X 0,Y 410.518,Z 309.388,A -85,B 0,C 180,E1 -11114.326,E2 -11114.326} C_VEL
LIN {X 0,Y 413.634,Z 176.425,A -85,B 0,C 180,E1 -11116.769,E2 -11116.769} C_VEL
LIN {X 0,Y 412.242,Z 172.308,A -85,B 0,C 180,E1 -11116.97,E2 -11116.97} C_VEL
LIN {X 0,Y 404.696,Z 156.275,A -85,B 0,C 180,E1 -11117.964,E2 -11117.964} C_VEL
LIN {X 0,Y 399.711,Z 146.264,A -85,B 0,C 180,E1 -11118.666,E2 -11118.666} C_VEL
LIN {X 0,Y 397.118,Z 136.652,A -85,B 0,C 180,E1 -11121.14,E2 -11121.14} C_VEL
LIN {X 0,Y 397.12,Z 136.639,A -85,B 0,C 180,E1 -11124.496,E2 -11124.496} C_VEL
LIN {X 0,Y 397.079,Z 136.64,A -85,B 0,C 180,E1 -11127.928,E2 -11127.928} C_VEL
LIN {X 0,Y 397.099,Z 136.635,A -85,B 0,C 180,E1 -11131.454,E2 -11131.454} C_VEL
LIN {X 0,Y 397.124,Z 136.637,A -85,B 0,C 180,E1 -11134.866,E2 -11134.866} C_VEL
LIN {X 0,Y 397.097,Z 136.648,A -85,B 0,C 180,E1 -11138.181,E2 -11138.181} C_VEL
LIN {X 0,Y 397.158,Z 136.64,A -85,B 0,C 180,E1 -11141.426,E2 -11141.426} C_VEL
LIN {X 0,Y 397.179,Z 136.631,A -85,B 0,C 180,E1 -11144.607,E2 -11144.607} C_VEL
LIN {X 0,Y 397.219,Z 136.628,A -85,B 0,C 180,E1 -11147.741,E2 -11147.741} C_VEL
LIN {X 0,Y 397.395,Z 136.609,A -85,B 0,C 180,E1 -11152.041,E2 -11152.041} C_VEL
LIN {X 0,Y 397.252,Z 136.619,A -85,B 0,C 180,E1 -11154.925,E2 -11154.925} C_VEL
LIN {X 0,Y 397.448,Z 136.596,A -85,B 0,C 180,E1 -11157.973,E2 -11157.973} C_VEL
LIN {X 0,Y 397.579,Z 136.585,A -85,B 0,C 180,E1 -11160,E2 -11160} C_VEL
LIN {X 0,Y 397.374,Z 136.611,A -85,B 0,C 180,E1 -11163.041,E2 -11163.041} C_VEL
LIN {X 0,Y 397.345,Z 136.612,A -85,B 0,C 180,E1 -11166.092,E2 -11166.092} C_VEL
LIN {X 0,Y 397.235,Z 136.624,A -85,B 0,C 180,E1 -11169.162,E2 -11169.162} C_VEL
LIN {X 0,Y 397.219,Z 136.625,A -85,B 0,C 180,E1 -11172.258,E2 -11172.258} C_VEL
LIN {X 0,Y 397.178,Z 136.63,A -85,B 0,C 180,E1 -11175.392,E2 -11175.392} C_VEL
LIN {X 0,Y 397.16,Z 136.639,A -85,B 0,C 180,E1 -11178.573,E2 -11178.573} C_VEL
LIN {X 0,Y 397.096,Z 136.644,A -85,B 0,C 180,E1 -11181.818,E2 -11181.818} C_VEL
LIN {X 0,Y 397.155,Z 136.637,A -85,B 0,C 180,E1 -11185.131,E2 -11185.131} C_VEL
LIN {X 0,Y 397.16,Z 136.637,A -85,B 0,C 180,E1 -11187.776,E2 -11187.776} C_VEL
LIN {X 0,Y 397.077,Z 136.649,A -85,B 0,C 180,E1 -11190.882,E2 -11190.882} C_VEL
LIN {X 0,Y 397.123,Z 136.641,A -85,B 0,C 180,E1 -11194.493,E2 -11194.493} C_VEL
LIN {X 0,Y 397.099,Z 136.632,A -85,B 0,C 180,E1 -11198.275,E2 -11198.275} C_VEL
LIN {X 0,Y 397.087,Z 136.649,A -85,B 0,C 180,E1 -11200.909,E2 -11200.909} C_VEL
LIN {X 0,Y 397.099,Z 136.634,A -85,B 0,C 180,E1 -11203.648,E2 -11203.648} C_VEL
LIN {X 0,Y 397.1,Z 136.636,A -85,B 0,C 180,E1 -11206.521,E2 -11206.521} C_VEL
LIN {X 0,Y 397.112,Z 136.639,A -85,B 0,C 180,E1 -11210.423,E2 -11210.423} C_VEL
LIN {X 0,Y 397.106,Z 136.645,A -85,B 0,C 180,E1 -11214.265,E2 -11214.265} C_VEL
LIN {X 0,Y 397.144,Z 136.813,A -85,B 0,C 180,E1 -11214.587,E2 -11214.587} C_VEL
LIN {X 0,Y 400.887,Z 149.981,A -85,B 0,C 180,E1 -11217.674,E2 -11217.674} C_VEL
LIN {X 0,Y 404.019,Z 162.662,A -85,B 0,C 180,E1 -11220.43,E2 -11220.43} C_VEL
LIN {X 0,Y 404.404,Z 164.647,A -85,B 0,C 180,E1 -11220.84,E2 -11220.84} C_VEL
LIN {X 0,Y 406.433,Z 169.766,A -85,B 0,C 180,E1 -11221.132,E2 -11221.132} C_VEL
LIN {X 0,Y 411.158,Z 191.411,A -85,B 0,C 180,E1 -11221.984,E2 -11221.984} C_VEL
LIN {X 0,Y 413.099,Z 203.012,A -85,B 0,C 180,E1 -11222.381,E2 -11222.381} C_VEL
LIN {X 0,Y 410.123,Z 331.073,A -85,B 0,C 180,E1 -11224.736,E2 -11224.736} C_VEL
LIN {X 0,Y 409.239,Z 347.022,A -85,B 0,C 180,E1 -11225.22,E2 -11225.22} C_VEL
LIN {X 0,Y 408.174,Z 361.092,A -85,B 0,C 180,E1 -11225.837,E2 -11225.837} C_VEL
LIN {X 0,Y 406.883,Z 374.333,A -85,B 0,C 180,E1 -11226.592,E2 -11226.592} C_VEL
LIN {X 0,Y 405.478,Z 388.045,A -85,B 0,C 180,E1 -11227.585,E2 -11227.585} C_VEL
LIN {X 0,Y 403.924,Z 400.667,A -85,B 0,C 180,E1 -11228.703,E2 -11228.703} C_VEL
LIN {X 0,Y 402.311,Z 413.464,A -85,B 0,C 180,E1 -11230.084,E2 -11230.084} C_VEL
LIN {X 0,Y 400.762,Z 425.117,A -85,B 0,C 180,E1 -11231.6,E2 -11231.6} C_VEL
LIN {X 0,Y 399.48,Z 434.951,A -85,B 0,C 180,E1 -11233.125,E2 -11233.125} C_VEL
LIN {X 0,Y 398.289,Z 444.608,A -85,B 0,C 180,E1 -11234.914,E2 -11234.914} C_VEL
LIN {X 0,Y 397.243,Z 453.246,A -85,B 0,C 180,E1 -11236.848,E2 -11236.848} C_VEL
LIN {X 0,Y 396.666,Z 460.244,A -85,B 0,C 180,E1 -11238.762,E2 -11238.762} C_VEL
LIN {X 0,Y 396.136,Z 466.28,A -85,B 0,C 180,E1 -11240.812,E2 -11240.812} C_VEL
LIN {X 0,Y 395.898,Z 470.938,A -85,B 0,C 180,E1 -11242.862,E2 -11242.862} C_VEL
LIN {X 0,Y 395.752,Z 474.305,A -85,B 0,C 180,E1 -11244.906,E2 -11244.906} C_VEL
LIN {X 0,Y 395.702,Z 476.474,A -85,B 0,C 180,E1 -11246.946,E2 -11246.946} C_VEL
LIN {X 0,Y 395.787,Z 477.495,A -85,B 0,C 180,E1 -11248.983,E2 -11248.983} C_VEL
LIN {X 0,Y 395.787,Z 477.376,A -85,B 0,C 180,E1 -11251.018,E2 -11251.018} C_VEL
LIN {X 0,Y 395.705,Z 476.08,A -85,B 0,C 180,E1 -11253.055,E2 -11253.055} C_VEL
LIN {X 0,Y 395.771,Z 473.569,A -85,B 0,C 180,E1 -11255.094,E2 -11255.094} C_VEL
LIN {X 0,Y 395.905,Z 469.829,A -85,B 0,C 180,E1 -11257.139,E2 -11257.139} C_VEL
LIN {X 0,Y 396.073,Z 464.757,A -85,B 0,C 180,E1 -11259.19,E2 -11259.19} C_VEL
LIN {X 0,Y 396.562,Z 458.227,A -85,B 0,C 180,E1 -11261.242,E2 -11261.242} C_VEL
LIN {X 0,Y 397.146,Z 450.161,A -85,B 0,C 180,E1 -11263.272,E2 -11263.272} C_VEL
LIN {X 0,Y 398.059,Z 441.295,A -85,B 0,C 180,E1 -11265.096,E2 -11265.096} C_VEL
LIN {X 0,Y 399.18,Z 430.752,A -85,B 0,C 180,E1 -11266.888,E2 -11266.888} C_VEL
LIN {X 0,Y 400.366,Z 419.929,A -85,B 0,C 180,E1 -11268.42,E2 -11268.42} C_VEL
LIN {X 0,Y 401.577,Z 408.107,A -85,B 0,C 180,E1 -11269.821,E2 -11269.821} C_VEL
LIN {X 0,Y 402.997,Z 395.202,A -85,B 0,C 180,E1 -11271.081,E2 -11271.081} C_VEL
LIN {X 0,Y 404.166,Z 382.735,A -85,B 0,C 180,E1 -11272.089,E2 -11272.089} C_VEL
LIN {X 0,Y 405.416,Z 368.466,A -85,B 0,C 180,E1 -11273.013,E2 -11273.013} C_VEL
LIN {X 0,Y 406.483,Z 353.212,A -85,B 0,C 180,E1 -11273.771,E2 -11273.771} C_VEL
LIN {X 0,Y 407.304,Z 338.601,A -85,B 0,C 180,E1 -11274.295,E2 -11274.295} C_VEL
LIN {X 0,Y 407.828,Z 322.427,A -85,B 0,C 180,E1 -11274.668,E2 -11274.668} C_VEL
LIN {X 0,Y 410.14,Z 202.094,A -85,B 0,C 180,E1 -11276.818,E2 -11276.818} C_VEL
LIN {X 0,Y 403.397,Z 165.199,A -85,B 0,C 180,E1 -11277.978,E2 -11277.978} C_VEL
LIN {X 0,Y 403.029,Z 161.508,A -85,B 0,C 180,E1 -11278.656,E2 -11278.656} C_VEL
LIN {X 0,Y 399.603,Z 146.784,A -85,B 0,C 180,E1 -11281.549,E2 -11281.549} C_VEL
LIN {X 0,Y 397.111,Z 136.65,A -85,B 0,C 180,E1 -11283.628,E2 -11283.628} C_VEL
LIN {X 0,Y 397.102,Z 136.649,A -85,B 0,C 180,E1 -11286.995,E2 -11286.995} C_VEL
LIN {X 0,Y 397.114,Z 136.647,A -85,B 0,C 180,E1 -11289.578,E2 -11289.578} C_VEL
LIN {X 0,Y 397.102,Z 136.65,A -85,B 0,C 180,E1 -11293.649,E2 -11293.649} C_VEL
LIN {X 0,Y 397.104,Z 136.646,A -85,B 0,C 180,E1 -11296.522,E2 -11296.522} C_VEL
LIN {X 0,Y 397.114,Z 136.638,A -85,B 0,C 180,E1 -11300.423,E2 -11300.423} C_VEL
LIN {X 0,Y 397.11,Z 136.64,A -85,B 0,C 180,E1 -11304.266,E2 -11304.266} C_VEL
LIN {X 0,Y 397.117,Z 136.642,A -85,B 0,C 180,E1 -11306.728,E2 -11306.728} C_VEL
LIN {X 0,Y 397.12,Z 136.638,A -85,B 0,C 180,E1 -11310.296,E2 -11310.296} C_VEL
LIN {X 0,Y 397.091,Z 136.637,A -85,B 0,C 180,E1 -11313.739,E2 -11313.739} C_VEL
LIN {X 0,Y 397.112,Z 136.642,A -85,B 0,C 180,E1 -11317.086,E2 -11317.086} C_VEL
LIN {X 0,Y 397.15,Z 136.637,A -85,B 0,C 180,E1 -11320.353,E2 -11320.353} C_VEL
LIN {X 0,Y 397.17,Z 136.63,A -85,B 0,C 180,E1 -11323.554,E2 -11323.554} C_VEL
LIN {X 0,Y 397.233,Z 136.627,A -85,B 0,C 180,E1 -11326.703,E2 -11326.703} C_VEL
LIN {X 0,Y 397.22,Z 136.628,A -85,B 0,C 180,E1 -11329.809,E2 -11329.809} C_VEL
LIN {X 0,Y 397.298,Z 136.618,A -85,B 0,C 180,E1 -11332.887,E2 -11332.887} C_VEL
LIN {X 0,Y 397.236,Z 136.626,A -85,B 0,C 180,E1 -11334.925,E2 -11334.925} C_VEL
LIN {X 0,Y 397.444,Z 136.589,A -85,B 0,C 180,E1 -11337.974,E2 -11337.974} C_VEL
LIN {X 0,Y 397.442,Z 136.593,A -85,B 0,C 180,E1 -11342.027,E2 -11342.027} C_VEL
LIN {X 0,Y 397.299,Z 136.612,A -85,B 0,C 180,E1 -11346.478,E2 -11346.478} C_VEL
LIN {X 0,Y 397.231,Z 136.605,A -85,B 0,C 180,E1 -11349.163,E2 -11349.163} C_VEL
LIN {X 0,Y 397.211,Z 136.627,A -85,B 0,C 180,E1 -11352.259,E2 -11352.259} C_VEL
LIN {X 0,Y 397.113,Z 136.643,A -85,B 0,C 180,E1 -11355.395,E2 -11355.395} C_VEL
LIN {X 0,Y 397.077,Z 136.644,A -85,B 0,C 180,E1 -11358.578,E2 -11358.578} C_VEL
LIN {X 0,Y 397.09,Z 136.642,A -85,B 0,C 180,E1 -11361.819,E2 -11361.819} C_VEL
LIN {X 0,Y 397.106,Z 136.646,A -85,B 0,C 180,E1 -11365.136,E2 -11365.136} C_VEL
LIN {X 0,Y 397.065,Z 136.633,A -85,B 0,C 180,E1 -11368.549,E2 -11368.549} C_VEL
LIN {X 0,Y 397.079,Z 136.642,A -85,B 0,C 180,E1 -11371.835,E2 -11371.835} C_VEL
LIN {X 0,Y 397.12,Z 136.641,A -85,B 0,C 180,E1 -11374.494,E2 -11374.494} C_VEL
LIN {X 0,Y 397.094,Z 136.624,A -85,B 0,C 180,E1 -11378.277,E2 -11378.277} C_VEL
LIN {X 0,Y 397.056,Z 136.648,A -85,B 0,C 180,E1 -11381.976,E2 -11381.976} C_VEL
LIN {X 0,Y 397.089,Z 136.632,A -85,B 0,C 180,E1 -11385.069,E2 -11385.069} C_VEL
LIN {X 0,Y 397.056,Z 136.646,A -85,B 0,C 180,E1 -11388.024,E2 -11388.024} C_VEL
LIN {X 0,Y 397.096,Z 136.636,A -85,B 0,C 180,E1 -11391.724,E2 -11391.724} C_VEL
LIN {X 0,Y 397.125,Z 136.64,A -85,B 0,C 180,E1 -11395.506,E2 -11395.506} C_VEL
LIN {X 0,Y 397.083,Z 136.647,A -85,B 0,C 180,E1 -11399.117,E2 -11399.117} C_VEL
LIN {X 0,Y 397.084,Z 136.646,A -85,B 0,C 180,E1 -11402.247,E2 -11402.247} C_VEL
LIN {X 0,Y 397.117,Z 136.648,A -85,B 0,C 180,E1 -11405.98,E2 -11405.98} C_VEL
LIN {X 0,Y 397.145,Z 136.641,A -85,B 0,C 180,E1 -11409.704,E2 -11409.704} C_VEL
LIN {X 0,Y 397.188,Z 136.622,A -85,B 0,C 180,E1 -11412.845,E2 -11412.845} C_VEL
LIN {X 0,Y 397.234,Z 136.62,A -85,B 0,C 180,E1 -11416.702,E2 -11416.702} C_VEL
LIN {X 0,Y 397.251,Z 136.757,A -85,B 0,C 180,E1 -11418.875,E2 -11418.875} C_VEL
LIN {X 0,Y 399.338,Z 145.683,A -85,B 0,C 180,E1 -11420.847,E2 -11420.847} C_VEL
LIN {X 0,Y 409.462,Z 170.5,A -85,B 0,C 180,E1 -11421.994,E2 -11421.994} C_VEL
LIN {X 0,Y 410.498,Z 176.17,A -85,B 0,C 180,E1 -11422.167,E2 -11422.167} C_VEL
LIN {X 0,Y 407.887,Z 310.447,A -85,B 0,C 180,E1 -11424.593,E2 -11424.593} C_VEL
LIN {X 0,Y 407.208,Z 326.334,A -85,B 0,C 180,E1 -11425.08,E2 -11425.08} C_VEL
LIN {X 0,Y 406.367,Z 340.812,A -85,B 0,C 180,E1 -11425.722,E2 -11425.722} C_VEL
LIN {X 0,Y 405.36,Z 354.479,A -85,B 0,C 180,E1 -11426.521,E2 -11426.521} C_VEL
LIN {X 0,Y 405.143,Z 357.325,A -85,B 0,C 180,E1 -11426.714,E2 -11426.714} C_VEL
LIN {X 0,Y 404.11,Z 362.646,A -85,B 0,C 180,E1 -11427.061,E2 -11427.061} C_VEL
LIN {X 0,Y 400.596,Z 371.085,A -85,B 0,C 180,E1 -11427.6,E2 -11427.6} C_VEL
LIN {X 0,Y 396.983,Z 379.293,A -85,B 0,C 180,E1 -11428.208,E2 -11428.208} C_VEL
LIN {X 0,Y 395.775,Z 384.101,A -85,B 0,C 180,E1 -11428.671,E2 -11428.671} C_VEL
LIN {X 0,Y 394.585,Z 395.577,A -85,B 0,C 180,E1 -11430,E2 -11430} C_VEL
LIN {X 0,Y 393.268,Z 406.694,A -85,B 0,C 180,E1 -11431.535,E2 -11431.535} C_VEL
LIN {X 0,Y 391.99,Z 417.516,A -85,B 0,C 180,E1 -11433.34,E2 -11433.34} C_VEL
LIN {X 0,Y 391.007,Z 426.518,A -85,B 0,C 180,E1 -11435.156,E2 -11435.156} C_VEL
LIN {X 0,Y 390.142,Z 434.971,A -85,B 0,C 180,E1 -11437.244,E2 -11437.244} C_VEL
LIN {X 0,Y 389.431,Z 441.799,A -85,B 0,C 180,E1 -11439.347,E2 -11439.347} C_VEL
LIN {X 0,Y 389.053,Z 447.15,A -85,B 0,C 180,E1 -11441.461,E2 -11441.461} C_VEL
LIN {X 0,Y 388.711,Z 451.159,A -85,B 0,C 180,E1 -11443.594,E2 -11443.594} C_VEL
LIN {X 0,Y 388.559,Z 453.87,A -85,B 0,C 180,E1 -11445.742,E2 -11445.742} C_VEL
LIN {X 0,Y 388.485,Z 455.345,A -85,B 0,C 180,E1 -11447.911,E2 -11447.911} C_VEL
LIN {X 0,Y 388.519,Z 455.577,A -85,B 0,C 180,E1 -11450.102,E2 -11450.102} C_VEL
LIN {X 0,Y 388.587,Z 454.535,A -85,B 0,C 180,E1 -11452.321,E2 -11452.321} C_VEL
LIN {X 0,Y 388.792,Z 452.152,A -85,B 0,C 180,E1 -11454.567,E2 -11454.567} C_VEL
LIN {X 0,Y 389.198,Z 448.33,A -85,B 0,C 180,E1 -11456.836,E2 -11456.836} C_VEL
LIN {X 0,Y 389.712,Z 442.925,A -85,B 0,C 180,E1 -11459.138,E2 -11459.138} C_VEL
LIN {X 0,Y 390.348,Z 437.745,A -85,B 0,C 180,E1 -11460.872,E2 -11460.872} C_VEL
LIN {X 0,Y 391.339,Z 430.263,A -85,B 0,C 180,E1 -11462.905,E2 -11462.905} C_VEL
LIN {X 0,Y 392.436,Z 422.384,A -85,B 0,C 180,E1 -11464.672,E2 -11464.672} C_VEL
LIN {X 0,Y 393.952,Z 411.935,A -85,B 0,C 180,E1 -11466.602,E2 -11466.602} C_VEL
LIN {X 0,Y 395.56,Z 400.832,A -85,B 0,C 180,E1 -11468.289,E2 -11468.289} C_VEL
LIN {X 0,Y 397.111,Z 389.365,A -85,B 0,C 180,E1 -11469.742,E2 -11469.742} C_VEL
LIN {X 0,Y 398.709,Z 376.985,A -85,B 0,C 180,E1 -11471.041,E2 -11471.041} C_VEL
LIN {X 0,Y 400.345,Z 363.417,A -85,B 0,C 180,E1 -11472.201,E2 -11472.201} C_VEL
LIN {X 0,Y 401.728,Z 348.953,A -85,B 0,C 180,E1 -11473.194,E2 -11473.194} C_VEL
LIN {X 0,Y 402.981,Z 333.575,A -85,B 0,C 180,E1 -11473.995,E2 -11473.995} C_VEL
LIN {X 0,Y 403.905,Z 319.007,A -85,B 0,C 180,E1 -11474.546,E2 -11474.546} C_VEL
LIN {X 0,Y 404.488,Z 303.335,A -85,B 0,C 180,E1 -11474.936,E2 -11474.936} C_VEL
LIN {X 0,Y 407.582,Z 177.831,A -85,B 0,C 180,E1 -11477.256,E2 -11477.256} C_VEL
LIN {X 0,Y 401.02,Z 163.241,A -85,B 0,C 180,E1 -11478.155,E2 -11478.155} C_VEL
LIN {X 0,Y 394.107,Z 149.746,A -85,B 0,C 180,E1 -11479.111,E2 -11479.111} C_VEL
LIN {X 0,Y 392.532,Z 146.453,A -85,B 0,C 180,E1 -11479.376,E2 -11479.376} C_VEL
LIN {X 0,Y 390.061,Z 137.525,A -85,B 0,C 180,E1 -11481.73,E2 -11481.73} C_VEL
LIN {X 0,Y 390.086,Z 137.512,A -85,B 0,C 180,E1 -11484.793,E2 -11484.793} C_VEL
LIN {X 0,Y 390.024,Z 137.519,A -85,B 0,C 180,E1 -11488.495,E2 -11488.495} C_VEL
LIN {X 0,Y 390.075,Z 137.509,A -85,B 0,C 180,E1 -11492.066,E2 -11492.066} C_VEL
LIN {X 0,Y 390.061,Z 137.509,A -85,B 0,C 180,E1 -11495.517,E2 -11495.517} C_VEL
LIN {X 0,Y 390.056,Z 137.521,A -85,B 0,C 180,E1 -11498.877,E2 -11498.877} C_VEL
LIN {X 0,Y 390.112,Z 137.513,A -85,B 0,C 180,E1 -11502.165,E2 -11502.165} C_VEL
LIN {X 0,Y 390.144,Z 137.508,A -85,B 0,C 180,E1 -11505.392,E2 -11505.392} C_VEL
LIN {X 0,Y 390.148,Z 137.508,A -85,B 0,C 180,E1 -11508.571,E2 -11508.571} C_VEL
LIN {X 0,Y 390.344,Z 137.486,A -85,B 0,C 180,E1 -11511.993,E2 -11511.993} C_VEL
LIN {X 0,Y 390.224,Z 137.494,A -85,B 0,C 180,E1 -11514.833,E2 -11514.833} C_VEL
LIN {X 0,Y 390.417,Z 137.472,A -85,B 0,C 180,E1 -11517.936,E2 -11517.936} C_VEL
LIN {X 0,Y 390.548,Z 137.461,A -85,B 0,C 180,E1 -11520,E2 -11520} C_VEL
LIN {X 0,Y 390.309,Z 137.491,A -85,B 0,C 180,E1 -11523.096,E2 -11523.096} C_VEL
LIN {X 0,Y 390.299,Z 137.489,A -85,B 0,C 180,E1 -11526.202,E2 -11526.202} C_VEL
LIN {X 0,Y 390.192,Z 137.502,A -85,B 0,C 180,E1 -11529.329,E2 -11529.329} C_VEL
LIN {X 0,Y 390.17,Z 137.503,A -85,B 0,C 180,E1 -11532.483,E2 -11532.483} C_VEL
LIN {X 0,Y 390.138,Z 137.505,A -85,B 0,C 180,E1 -11535.676,E2 -11535.676} C_VEL
LIN {X 0,Y 390.104,Z 137.514,A -85,B 0,C 180,E1 -11538.922,E2 -11538.922} C_VEL
LIN {X 0,Y 390.039,Z 137.524,A -85,B 0,C 180,E1 -11542.234,E2 -11542.234} C_VEL
LIN {X 0,Y 390.118,Z 137.511,A -85,B 0,C 180,E1 -11545.743,E2 -11545.743} C_VEL
LIN {X 0,Y 390.057,Z 137.518,A -85,B 0,C 180,E1 -11549.109,E2 -11549.109} C_VEL
LIN {X 0,Y 390.041,Z 137.523,A -85,B 0,C 180,E1 -11552.721,E2 -11552.721} C_VEL
LIN {X 0,Y 390.054,Z 137.522,A -85,B 0,C 180,E1 -11555.825,E2 -11555.825} C_VEL
LIN {X 0,Y 390.066,Z 137.508,A -85,B 0,C 180,E1 -11559.218,E2 -11559.218} C_VEL
LIN {X 0,Y 390.04,Z 137.515,A -85,B 0,C 180,E1 -11562.374,E2 -11562.374} C_VEL
LIN {X 0,Y 390.042,Z 137.525,A -85,B 0,C 180,E1 -11565.354,E2 -11565.354} C_VEL
LIN {X 0,Y 390.029,Z 137.527,A -85,B 0,C 180,E1 -11568.187,E2 -11568.187} C_VEL
LIN {X 0,Y 390.089,Z 137.518,A -85,B 0,C 180,E1 -11570.908,E2 -11570.908} C_VEL
LIN {X 0,Y 390.055,Z 137.594,A -85,B 0,C 180,E1 -11573.936,E2 -11573.936} C_VEL
LIN {X 0,Y 393.473,Z 149.482,A -85,B 0,C 180,E1 -11576.828,E2 -11576.828} C_VEL
LIN {X 0,Y 396.724,Z 162.117,A -85,B 0,C 180,E1 -11579.678,E2 -11579.678} C_VEL
LIN {X 0,Y 397.229,Z 164.397,A -85,B 0,C 180,E1 -11580.168,E2 -11580.168} C_VEL
LIN {X 0,Y 400.744,Z 172.589,A -85,B 0,C 180,E1 -11580.675,E2 -11580.675} C_VEL
LIN {X 0,Y 405.358,Z 194.192,A -85,B 0,C 180,E1 -11581.546,E2 -11581.546} C_VEL
LIN {X 0,Y 407.006,Z 203.632,A -85,B 0,C 180,E1 -11581.884,E2 -11581.884} C_VEL
LIN {X 0,Y 403.896,Z 330.431,A -85,B 0,C 180,E1 -11584.249,E2 -11584.249} C_VEL
LIN {X 0,Y 402.954,Z 346.57,A -85,B 0,C 180,E1 -11584.738,E2 -11584.738} C_VEL
LIN {X 0,Y 401.872,Z 360.502,A -85,B 0,C 180,E1 -11585.355,E2 -11585.355} C_VEL
LIN {X 0,Y 400.415,Z 374.957,A -85,B 0,C 180,E1 -11586.191,E2 -11586.191} C_VEL
LIN {X 0,Y 398.951,Z 388.501,A -85,B 0,C 180,E1 -11587.198,E2 -11587.198} C_VEL
LIN {X 0,Y 397.322,Z 401.003,A -85,B 0,C 180,E1 -11588.331,E2 -11588.331} C_VEL
LIN {X 0,Y 395.638,Z 413.708,A -85,B 0,C 180,E1 -11589.734,E2 -11589.734} C_VEL
LIN {X 0,Y 394.005,Z 425.27,A -85,B 0,C 180,E1 -11591.273,E2 -11591.273} C_VEL
LIN {X 0,Y 392.64,Z 435.029,A -85,B 0,C 180,E1 -11592.822,E2 -11592.822} C_VEL
LIN {X 0,Y 391.379,Z 444.627,A -85,B 0,C 180,E1 -11594.641,E2 -11594.641} C_VEL
LIN {X 0,Y 390.239,Z 452.943,A -85,B 0,C 180,E1 -11596.534,E2 -11596.534} C_VEL
LIN {X 0,Y 389.634,Z 460.187,A -85,B 0,C 180,E1 -11598.556,E2 -11598.556} C_VEL
LIN {X 0,Y 389.062,Z 466.19,A -85,B 0,C 180,E1 -11600.644,E2 -11600.644} C_VEL
LIN {X 0,Y 388.818,Z 470.83,A -85,B 0,C 180,E1 -11602.731,E2 -11602.731} C_VEL
LIN {X 0,Y 388.658,Z 474.168,A -85,B 0,C 180,E1 -11604.813,E2 -11604.813} C_VEL
LIN {X 0,Y 388.609,Z 476.308,A -85,B 0,C 180,E1 -11606.89,E2 -11606.89} C_VEL
LIN {X 0,Y 388.699,Z 477.302,A -85,B 0,C 180,E1 -11608.964,E2 -11608.964} C_VEL
LIN {X 0,Y 388.699,Z 477.157,A -85,B 0,C 180,E1 -11611.036,E2 -11611.036} C_VEL
LIN {X 0,Y 388.612,Z 475.846,A -85,B 0,C 180,E1 -11613.111,E2 -11613.111} C_VEL
LIN {X 0,Y 388.676,Z 473.309,A -85,B 0,C 180,E1 -11615.188,E2 -11615.188} C_VEL
LIN {X 0,Y 388.823,Z 469.537,A -85,B 0,C 180,E1 -11617.269,E2 -11617.269} C_VEL
LIN {X 0,Y 389.009,Z 464.429,A -85,B 0,C 180,E1 -11619.358,E2 -11619.358} C_VEL
LIN {X 0,Y 389.536,Z 457.857,A -85,B 0,C 180,E1 -11621.447,E2 -11621.447} C_VEL
LIN {X 0,Y 390.077,Z 450.387,A -85,B 0,C 180,E1 -11623.366,E2 -11623.366} C_VEL
LIN {X 0,Y 390.972,Z 442.202,A -85,B 0,C 180,E1 -11625.109,E2 -11625.109} C_VEL
LIN {X 0,Y 391.893,Z 433.513,A -85,B 0,C 180,E1 -11626.675,E2 -11626.675} C_VEL
LIN {X 0,Y 393.098,Z 423.215,A -85,B 0,C 180,E1 -11628.233,E2 -11628.233} C_VEL
LIN {X 0,Y 394.435,Z 410.948,A -85,B 0,C 180,E1 -11629.788,E2 -11629.788} C_VEL
LIN {X 0,Y 395.831,Z 398.64,A -85,B 0,C 180,E1 -11631.072,E2 -11631.072} C_VEL
LIN {X 0,Y 397.163,Z 385.233,A -85,B 0,C 180,E1 -11632.225,E2 -11632.225} C_VEL
LIN {X 0,Y 398.479,Z 371.771,A -85,B 0,C 180,E1 -11633.153,E2 -11633.153} C_VEL
LIN {X 0,Y 399.592,Z 357.463,A -85,B 0,C 180,E1 -11633.931,E2 -11633.931} C_VEL
LIN {X 0,Y 400.475,Z 342.657,A -85,B 0,C 180,E1 -11634.529,E2 -11634.529} C_VEL
LIN {X 0,Y 401.112,Z 327.673,A -85,B 0,C 180,E1 -11634.937,E2 -11634.937} C_VEL
LIN {X 0,Y 403.627,Z 203.45,A -85,B 0,C 180,E1 -11637.198,E2 -11637.198} C_VEL
LIN {X 0,Y 398.633,Z 175.23,A -85,B 0,C 180,E1 -11638.075,E2 -11638.075} C_VEL
LIN {X 0,Y 396.546,Z 165.072,A -85,B 0,C 180,E1 -11638.428,E2 -11638.428} C_VEL
LIN {X 0,Y 393.448,Z 151.054,A -85,B 0,C 180,E1 -11641.2,E2 -11641.2} C_VEL
LIN {X 0,Y 390.07,Z 137.525,A -85,B 0,C 180,E1 -11644.025,E2 -11644.025} C_VEL
LIN {X 0,Y 390.045,Z 137.527,A -85,B 0,C 180,E1 -11647.551,E2 -11647.551} C_VEL
LIN {X 0,Y 390.056,Z 137.523,A -85,B 0,C 180,E1 -11650.822,E2 -11650.822} C_VEL
LIN {X 0,Y 390.056,Z 137.526,A -85,B 0,C 180,E1 -11653.887,E2 -11653.887} C_VEL
LIN {X 0,Y 390.059,Z 137.525,A -85,B 0,C 180,E1 -11656.79,E2 -11656.79} C_VEL
LIN {X 0,Y 390.058,Z 137.523,A -85,B 0,C 180,E1 -11659.561,E2 -11659.561} C_VEL
LIN {X 0,Y 390.044,Z 137.521,A -85,B 0,C 180,E1 -11662.45,E2 -11662.45} C_VEL
LIN {X 0,Y 390.071,Z 137.519,A -85,B 0,C 180,E1 -11665.976,E2 -11665.976} C_VEL
LIN {X 0,Y 390.04,Z 137.521,A -85,B 0,C 180,E1 -11669.701,E2 -11669.701} C_VEL
LIN {X 0,Y 390.049,Z 137.508,A -85,B 0,C 180,E1 -11673.227,E2 -11673.227} C_VEL
LIN {X 0,Y 390.081,Z 137.521,A -85,B 0,C 180,E1 -11676.761,E2 -11676.761} C_VEL
LIN {X 0,Y 390.107,Z 137.513,A -85,B 0,C 180,E1 -11679.984,E2 -11679.984} C_VEL
LIN {X 0,Y 390.142,Z 137.507,A -85,B 0,C 180,E1 -11683.249,E2 -11683.249} C_VEL
LIN {X 0,Y 390.199,Z 137.505,A -85,B 0,C 180,E1 -11686.562,E2 -11686.562} C_VEL
LIN {X 0,Y 390.171,Z 137.506,A -85,B 0,C 180,E1 -11689.623,E2 -11689.623} C_VEL
LIN {X 0,Y 390.251,Z 137.496,A -85,B 0,C 180,E1 -11692.758,E2 -11692.758} C_VEL
LIN {X 0,Y 390.207,Z 137.503,A -85,B 0,C 180,E1 -11694.834,E2 -11694.834} C_VEL
LIN {X 0,Y 390.412,Z 137.465,A -85,B 0,C 180,E1 -11697.937,E2 -11697.937} C_VEL
LIN {X 0,Y 390.408,Z 137.469,A -85,B 0,C 180,E1 -11702.064,E2 -11702.064} C_VEL
LIN {X 0,Y 390.26,Z 137.489,A -85,B 0,C 180,E1 -11706.47,E2 -11706.47} C_VEL
LIN {X 0,Y 390.189,Z 137.48,A -85,B 0,C 180,E1 -11709.33,E2 -11709.33} C_VEL
LIN {X 0,Y 390.158,Z 137.504,A -85,B 0,C 180,E1 -11712.484,E2 -11712.484} C_VEL
LIN {X 0,Y 390.057,Z 137.522,A -85,B 0,C 180,E1 -11715.681,E2 -11715.681} C_VEL
LIN {X 0,Y 390.035,Z 137.522,A -85,B 0,C 180,E1 -11718.926,E2 -11718.926} C_VEL
LIN {X 0,Y 390.033,Z 137.519,A -85,B 0,C 180,E1 -11722.235,E2 -11722.235} C_VEL
LIN {X 0,Y 390.055,Z 137.52,A -85,B 0,C 180,E1 -11725.722,E2 -11725.722} C_VEL
LIN {X 0,Y 390.026,Z 137.504,A -85,B 0,C 180,E1 -11729.113,E2 -11729.113} C_VEL
LIN {X 0,Y 390.043,Z 137.519,A -85,B 0,C 180,E1 -11732.722,E2 -11732.722} C_VEL
LIN {X 0,Y 390.046,Z 137.516,A -85,B 0,C 180,E1 -11735.822,E2 -11735.822} C_VEL
LIN {X 0,Y 390.04,Z 137.509,A -85,B 0,C 180,E1 -11739.212,E2 -11739.212} C_VEL
LIN {X 0,Y 390.035,Z 137.524,A -85,B 0,C 180,E1 -11742.372,E2 -11742.372} C_VEL
LIN {X 0,Y 390.045,Z 137.506,A -85,B 0,C 180,E1 -11745.354,E2 -11745.354} C_VEL
LIN {X 0,Y 390.02,Z 137.523,A -85,B 0,C 180,E1 -11748.184,E2 -11748.184} C_VEL
LIN {X 0,Y 390.062,Z 137.515,A -85,B 0,C 180,E1 -11750.904,E2 -11750.904} C_VEL
LIN {X 0,Y 390.087,Z 137.52,A -85,B 0,C 180,E1 -11754.793,E2 -11754.793} C_VEL
LIN {X 0,Y 390.028,Z 137.524,A -85,B 0,C 180,E1 -11758.495,E2 -11758.495} C_VEL
LIN {X 0,Y 390.03,Z 137.523,A -85,B 0,C 180,E1 -11762.063,E2 -11762.063} C_VEL
LIN {X 0,Y 390.048,Z 137.526,A -85,B 0,C 180,E1 -11765.517,E2 -11765.517} C_VEL
LIN {X 0,Y 390.061,Z 137.521,A -85,B 0,C 180,E1 -11768.878,E2 -11768.878} C_VEL
LIN {X 0,Y 390.116,Z 137.5,A -85,B 0,C 180,E1 -11772.166,E2 -11772.166} C_VEL
LIN {X 0,Y 390.149,Z 137.506,A -85,B 0,C 180,E1 -11775.392,E2 -11775.392} C_VEL
LIN {X 0,Y 390.201,Z 137.678,A -85,B 0,C 180,E1 -11778.506,E2 -11778.506} C_VEL
LIN {X 0,Y 392.117,Z 145.829,A -85,B 0,C 180,E1 -11780.352,E2 -11780.352} C_VEL
LIN {X 0,Y 403.164,Z 172.552,A -85,B 0,C 180,E1 -11781.63,E2 -11781.63} C_VEL
LIN {X 0,Y 404.02,Z 176.775,A -85,B 0,C 180,E1 -11781.768,E2 -11781.768} C_VEL
LIN {X 0,Y 401.315,Z 310.598,A -85,B 0,C 180,E1 -11784.22,E2 -11784.22} C_VEL
LIN {X 0,Y 400.65,Z 325.695,A -85,B 0,C 180,E1 -11784.684,E2 -11784.684} C_VEL
LIN {X 0,Y 399.777,Z 340.383,A -85,B 0,C 180,E1 -11785.336,E2 -11785.336} C_VEL
LIN {X 0,Y 398.667,Z 355.175,A -85,B 0,C 180,E1 -11786.209,E2 -11786.209} C_VEL
LIN {X 0,Y 397.448,Z 368.55,A -85,B 0,C 180,E1 -11787.212,E2 -11787.212} C_VEL
LIN {X 0,Y 396.026,Z 382.208,A -85,B 0,C 180,E1 -11788.474,E2 -11788.474} C_VEL
LIN {X 0,Y 395.775,Z 384.101,A -85,B 0,C 180,E1 -11788.671,E2 -11788.671} C_VEL
LIN {X 0,Y 394.584,Z 388.865,A -85,B 0,C 180,E1 -11789.158,E2 -11789.158} C_VEL
LIN {X 0,Y 387.974,Z 402.167,A -85,B 0,C 180,E1 -11790.609,E2 -11790.609} C_VEL
LIN {X 0,Y 386.519,Z 406.35,A -85,B 0,C 180,E1 -11791.187,E2 -11791.187} C_VEL
LIN {X 0,Y 386.296,Z 407.695,A -85,B 0,C 180,E1 -11791.397,E2 -11791.397} C_VEL
LIN {X 0,Y 385.049,Z 417.892,A -85,B 0,C 180,E1 -11793.138,E2 -11793.138} C_VEL
LIN {X 0,Y 384.004,Z 426.871,A -85,B 0,C 180,E1 -11794.987,E2 -11794.987} C_VEL
LIN {X 0,Y 383.166,Z 434.347,A -85,B 0,C 180,E1 -11796.847,E2 -11796.847} C_VEL
LIN {X 0,Y 382.62,Z 439.702,A -85,B 0,C 180,E1 -11798.45,E2 -11798.45} C_VEL
LIN {X 0,Y 382.092,Z 445.563,A -85,B 0,C 180,E1 -11800.599,E2 -11800.599} C_VEL
LIN {X 0,Y 381.762,Z 450.039,A -85,B 0,C 180,E1 -11802.762,E2 -11802.762} C_VEL
LIN {X 0,Y 381.487,Z 453.233,A -85,B 0,C 180,E1 -11804.946,E2 -11804.946} C_VEL
LIN {X 0,Y 381.405,Z 455.179,A -85,B 0,C 180,E1 -11807.147,E2 -11807.147} C_VEL
LIN {X 0,Y 381.418,Z 455.869,A -85,B 0,C 180,E1 -11809.37,E2 -11809.37} C_VEL
LIN {X 0,Y 381.432,Z 455.279,A -85,B 0,C 180,E1 -11811.623,E2 -11811.623} C_VEL
LIN {X 0,Y 381.609,Z 453.377,A -85,B 0,C 180,E1 -11813.901,E2 -11813.901} C_VEL
LIN {X 0,Y 382.021,Z 450.081,A -85,B 0,C 180,E1 -11816.201,E2 -11816.201} C_VEL
LIN {X 0,Y 382.498,Z 445.265,A -85,B 0,C 180,E1 -11818.536,E2 -11818.536} C_VEL
LIN {X 0,Y 383.135,Z 440.116,A -85,B 0,C 180,E1 -11820.441,E2 -11820.441} C_VEL
LIN {X 0,Y 384.038,Z 433.632,A -85,B 0,C 180,E1 -11822.387,E2 -11822.387} C_VEL
LIN {X 0,Y 385.214,Z 425.219,A -85,B 0,C 180,E1 -11824.442,E2 -11824.442} C_VEL
LIN {X 0,Y 386.619,Z 416.412,A -85,B 0,C 180,E1 -11826.213,E2 -11826.213} C_VEL
LIN {X 0,Y 388.174,Z 405.786,A -85,B 0,C 180,E1 -11827.994,E2 -11827.994} C_VEL
LIN {X 0,Y 389.953,Z 394.076,A -85,B 0,C 180,E1 -11829.609,E2 -11829.609} C_VEL
LIN {X 0,Y 391.603,Z 382.189,A -85,B 0,C 180,E1 -11830.974,E2 -11830.974} C_VEL
LIN {X 0,Y 393.139,Z 370.481,A -85,B 0,C 180,E1 -11832.096,E2 -11832.096} C_VEL
LIN {X 0,Y 394.815,Z 355.908,A -85,B 0,C 180,E1 -11833.225,E2 -11833.225} C_VEL
LIN {X 0,Y 396.176,Z 340.974,A -85,B 0,C 180,E1 -11834.129,E2 -11834.129} C_VEL
LIN {X 0,Y 397.296,Z 325.714,A -85,B 0,C 180,E1 -11834.815,E2 -11834.815} C_VEL
LIN {X 0,Y 398.092,Z 310.644,A -85,B 0,C 180,E1 -11835.28,E2 -11835.28} C_VEL
LIN {X 0,Y 401.442,Z 179.539,A -85,B 0,C 180,E1 -11837.767,E2 -11837.767} C_VEL
LIN {X 0,Y 392.736,Z 160.876,A -85,B 0,C 180,E1 -11839,E2 -11839} C_VEL
LIN {X 0,Y 385.374,Z 146.794,A -85,B 0,C 180,E1 -11840.08,E2 -11840.08} C_VEL
LIN {X 0,Y 383.023,Z 138.397,A -85,B 0,C 180,E1 -11842.375,E2 -11842.375} C_VEL
LIN {X 0,Y 383.019,Z 138.393,A -85,B 0,C 180,E1 -11845.659,E2 -11845.659} C_VEL
LIN {X 0,Y 382.983,Z 138.401,A -85,B 0,C 180,E1 -11849.081,E2 -11849.081} C_VEL
LIN {X 0,Y 383.019,Z 138.393,A -85,B 0,C 180,E1 -11852.695,E2 -11852.695} C_VEL
LIN {X 0,Y 383.017,Z 138.384,A -85,B 0,C 180,E1 -11856.191,E2 -11856.191} C_VEL
LIN {X 0,Y 383.056,Z 138.392,A -85,B 0,C 180,E1 -11859.598,E2 -11859.598} C_VEL
LIN {X 0,Y 383.094,Z 138.387,A -85,B 0,C 180,E1 -11862.93,E2 -11862.93} C_VEL
LIN {X 0,Y 383.126,Z 138.386,A -85,B 0,C 180,E1 -11866.463,E2 -11866.463} C_VEL
LIN {X 0,Y 383.152,Z 138.379,A -85,B 0,C 180,E1 -11870.497,E2 -11870.497} C_VEL
LIN {X 0,Y 383.272,Z 138.367,A -85,B 0,C 180,E1 -11872.625,E2 -11872.625} C_VEL
LIN {X 0,Y 383.197,Z 138.369,A -85,B 0,C 180,E1 -11874.738,E2 -11874.738} C_VEL
LIN {X 0,Y 383.385,Z 138.347,A -85,B 0,C 180,E1 -11877.898,E2 -11877.898} C_VEL
LIN {X 0,Y 383.518,Z 138.336,A -85,B 0,C 180,E1 -11880,E2 -11880} C_VEL
LIN {X 0,Y 383.245,Z 138.372,A -85,B 0,C 180,E1 -11883.153,E2 -11883.153} C_VEL
LIN {X 0,Y 383.256,Z 138.367,A -85,B 0,C 180,E1 -11886.316,E2 -11886.316} C_VEL
LIN {X 0,Y 383.142,Z 138.381,A -85,B 0,C 180,E1 -11889.502,E2 -11889.502} C_VEL
LIN {X 0,Y 383.124,Z 138.386,A -85,B 0,C 180,E1 -11893.536,E2 -11893.536} C_VEL
LIN {X 0,Y 383.093,Z 138.39,A -85,B 0,C 180,E1 -11897.454,E2 -11897.454} C_VEL
LIN {X 0,Y 383.028,Z 138.395,A -85,B 0,C 180,E1 -11900.647,E2 -11900.647} C_VEL
LIN {X 0,Y 383.032,Z 138.395,A -85,B 0,C 180,E1 -11903.807,E2 -11903.807} C_VEL
LIN {X 0,Y 383.055,Z 138.395,A -85,B 0,C 180,E1 -11907.302,E2 -11907.302} C_VEL
LIN {X 0,Y 382.981,Z 138.405,A -85,B 0,C 180,E1 -11910.918,E2 -11910.918} C_VEL
LIN {X 0,Y 383.016,Z 138.397,A -85,B 0,C 180,E1 -11914.668,E2 -11914.668} C_VEL
LIN {X 0,Y 382.997,Z 138.39,A -85,B 0,C 180,E1 -11917.903,E2 -11917.903} C_VEL
LIN {X 0,Y 382.982,Z 138.405,A -85,B 0,C 180,E1 -11921.347,E2 -11921.347} C_VEL
LIN {X 0,Y 382.994,Z 138.397,A -85,B 0,C 180,E1 -11924.303,E2 -11924.303} C_VEL
LIN {X 0,Y 383.008,Z 138.391,A -85,B 0,C 180,E1 -11927.24,E2 -11927.24} C_VEL
LIN {X 0,Y 383.013,Z 138.394,A -85,B 0,C 180,E1 -11930.413,E2 -11930.413} C_VEL
LIN {X 0,Y 383.023,Z 138.544,A -85,B 0,C 180,E1 -11933.299,E2 -11933.299} C_VEL
LIN {X 0,Y 386.525,Z 150.493,A -85,B 0,C 180,E1 -11936.3,E2 -11936.3} C_VEL
LIN {X 0,Y 389.501,Z 162.033,A -85,B 0,C 180,E1 -11938.988,E2 -11938.988} C_VEL
LIN {X 0,Y 390.098,Z 164.359,A -85,B 0,C 180,E1 -11939.472,E2 -11939.472} C_VEL
LIN {X 0,Y 395.07,Z 175.396,A -85,B 0,C 180,E1 -11940.201,E2 -11940.201} C_VEL
LIN {X 0,Y 399.41,Z 195.929,A -85,B 0,C 180,E1 -11941.053,E2 -11941.053} C_VEL
LIN {X 0,Y 400.942,Z 205.247,A -85,B 0,C 180,E1 -11941.388,E2 -11941.388} C_VEL
LIN {X 0,Y 397.73,Z 330.052,A -85,B 0,C 180,E1 -11943.749,E2 -11943.749} C_VEL
LIN {X 0,Y 396.744,Z 346.239,A -85,B 0,C 180,E1 -11944.244,E2 -11944.244} C_VEL
LIN {X 0,Y 395.58,Z 360.054,A -85,B 0,C 180,E1 -11944.859,E2 -11944.859} C_VEL
LIN {X 0,Y 394.199,Z 374.043,A -85,B 0,C 180,E1 -11945.68,E2 -11945.68} C_VEL
LIN {X 0,Y 392.642,Z 387.393,A -85,B 0,C 180,E1 -11946.671,E2 -11946.671} C_VEL
LIN {X 0,Y 390.883,Z 400.058,A -85,B 0,C 180,E1 -11947.817,E2 -11947.817} C_VEL
LIN {X 0,Y 389.101,Z 412.89,A -85,B 0,C 180,E1 -11949.239,E2 -11949.239} C_VEL
LIN {X 0,Y 387.4,Z 424.363,A -85,B 0,C 180,E1 -11950.774,E2 -11950.774} C_VEL
LIN {X 0,Y 385.828,Z 435.139,A -85,B 0,C 180,E1 -11952.51,E2 -11952.51} C_VEL
LIN {X 0,Y 384.484,Z 444.681,A -85,B 0,C 180,E1 -11954.359,E2 -11954.359} C_VEL
LIN {X 0,Y 383.203,Z 453.44,A -85,B 0,C 180,E1 -11956.416,E2 -11956.416} C_VEL
LIN {X 0,Y 382.614,Z 460.133,A -85,B 0,C 180,E1 -11958.343,E2 -11958.343} C_VEL
LIN {X 0,Y 382.008,Z 466.101,A -85,B 0,C 180,E1 -11960.47,E2 -11960.47} C_VEL
LIN {X 0,Y 381.726,Z 470.717,A -85,B 0,C 180,E1 -11962.596,E2 -11962.596} C_VEL
LIN {X 0,Y 381.57,Z 474.034,A -85,B 0,C 180,E1 -11964.716,E2 -11964.716} C_VEL
LIN {X 0,Y 381.519,Z 476.144,A -85,B 0,C 180,E1 -11966.832,E2 -11966.832} C_VEL
LIN {X 0,Y 381.613,Z 477.11,A -85,B 0,C 180,E1 -11968.945,E2 -11968.945} C_VEL
LIN {X 0,Y 381.614,Z 476.936,A -85,B 0,C 180,E1 -11971.056,E2 -11971.056} C_VEL
LIN {X 0,Y 381.523,Z 475.603,A -85,B 0,C 180,E1 -11973.168,E2 -11973.168} C_VEL
LIN {X 0,Y 381.586,Z 473.04,A -85,B 0,C 180,E1 -11975.284,E2 -11975.284} C_VEL
LIN {X 0,Y 381.727,Z 469.235,A -85,B 0,C 180,E1 -11977.405,E2 -11977.405} C_VEL
LIN {X 0,Y 381.955,Z 464.092,A -85,B 0,C 180,E1 -11979.533,E2 -11979.533} C_VEL
LIN {X 0,Y 382.51,Z 457.481,A -85,B 0,C 180,E1 -11981.661,E2 -11981.661} C_VEL
LIN {X 0,Y 383.047,Z 450.506,A -85,B 0,C 180,E1 -11983.488,E2 -11983.488} C_VEL
LIN {X 0,Y 384.033,Z 441.736,A -85,B 0,C 180,E1 -11985.389,E2 -11985.389} C_VEL
LIN {X 0,Y 385.237,Z 431.362,A -85,B 0,C 180,E1 -11987.245,E2 -11987.245} C_VEL
LIN {X 0,Y 386.563,Z 420.273,A -85,B 0,C 180,E1 -11988.892,E2 -11988.892} C_VEL
LIN {X 0,Y 387.794,Z 409.139,A -85,B 0,C 180,E1 -11990.28,E2 -11990.28} C_VEL
LIN {X 0,Y 389.306,Z 396.523,A -85,B 0,C 180,E1 -11991.582,E2 -11991.582} C_VEL
LIN {X 0,Y 390.741,Z 382.66,A -85,B 0,C 180,E1 -11992.75,E2 -11992.75} C_VEL
LIN {X 0,Y 392.072,Z 368.343,A -85,B 0,C 180,E1 -11993.71,E2 -11993.71} C_VEL
LIN {X 0,Y 393.198,Z 353.312,A -85,B 0,C 180,E1 -11994.485,E2 -11994.485} C_VEL
LIN {X 0,Y 394.158,Z 337.792,A -85,B 0,C 180,E1 -11995.055,E2 -11995.055} C_VEL
LIN {X 0,Y 394.677,Z 321.35,A -85,B 0,C 180,E1 -11995.442,E2 -11995.442} C_VEL
LIN {X 0,Y 397.088,Z 203.256,A -85,B 0,C 180,E1 -11997.62,E2 -11997.62} C_VEL
LIN {X 0,Y 390.455,Z 167.946,A -85,B 0,C 180,E1 -11998.774,E2 -11998.774} C_VEL
LIN {X 0,Y 389.354,Z 164.938,A -85,B 0,C 180,E1 -11998.912,E2 -11998.912} C_VEL
LIN {X 0,Y 386.004,Z 150.366,A -85,B 0,C 180,E1 -12001.871,E2 -12001.871} C_VEL
LIN {X 0,Y 383.017,Z 138.404,A -85,B 0,C 180,E1 -12004.459,E2 -12004.459} C_VEL
LIN {X 0,Y 383.001,Z 138.402,A -85,B 0,C 180,E1 -12007.904,E2 -12007.904} C_VEL
LIN {X 0,Y 382.983,Z 138.405,A -85,B 0,C 180,E1 -12011.348,E2 -12011.348} C_VEL
LIN {X 0,Y 382.997,Z 138.405,A -85,B 0,C 180,E1 -12014.304,E2 -12014.304} C_VEL
LIN {X 0,Y 383.012,Z 138.406,A -85,B 0,C 180,E1 -12017.241,E2 -12017.241} C_VEL
LIN {X 0,Y 383.015,Z 138.394,A -85,B 0,C 180,E1 -12020.415,E2 -12020.415} C_VEL
LIN {X 0,Y 383.027,Z 138.395,A -85,B 0,C 180,E1 -12024.045,E2 -12024.045} C_VEL
LIN {X 0,Y 382.989,Z 138.402,A -85,B 0,C 180,E1 -12027.579,E2 -12027.579} C_VEL
LIN {X 0,Y 382.981,Z 138.399,A -85,B 0,C 180,E1 -12030.3,E2 -12030.3} C_VEL
LIN {X 0,Y 383.006,Z 138.39,A -85,B 0,C 180,E1 -12034.045,E2 -12034.045} C_VEL
LIN {X 0,Y 383,Z 138.397,A -85,B 0,C 180,E1 -12037.335,E2 -12037.335} C_VEL
LIN {X 0,Y 383.062,Z 138.396,A -85,B 0,C 180,E1 -12040.717,E2 -12040.717} C_VEL
LIN {X 0,Y 383.083,Z 138.385,A -85,B 0,C 180,E1 -12044.027,E2 -12044.027} C_VEL
LIN {X 0,Y 383.141,Z 138.377,A -85,B 0,C 180,E1 -12047.284,E2 -12047.284} C_VEL
LIN {X 0,Y 383.147,Z 138.385,A -85,B 0,C 180,E1 -12050.498,E2 -12050.498} C_VEL
LIN {X 0,Y 383.243,Z 138.367,A -85,B 0,C 180,E1 -12053.683,E2 -12053.683} C_VEL
LIN {X 0,Y 383.377,Z 138.341,A -85,B 0,C 180,E1 -12057.899,E2 -12057.899} C_VEL
LIN {X 0,Y 383.373,Z 138.346,A -85,B 0,C 180,E1 -12062.102,E2 -12062.102} C_VEL
LIN {X 0,Y 383.226,Z 138.365,A -85,B 0,C 180,E1 -12066.458,E2 -12066.458} C_VEL
LIN {X 0,Y 383.14,Z 138.357,A -85,B 0,C 180,E1 -12069.503,E2 -12069.503} C_VEL
LIN {X 0,Y 383.114,Z 138.381,A -85,B 0,C 180,E1 -12072.717,E2 -12072.717} C_VEL
LIN {X 0,Y 383.006,Z 138.396,A -85,B 0,C 180,E1 -12075.977,E2 -12075.977} C_VEL
LIN {X 0,Y 383.004,Z 138.4,A -85,B 0,C 180,E1 -12079.287,E2 -12079.287} C_VEL
LIN {X 0,Y 382.987,Z 138.396,A -85,B 0,C 180,E1 -12082.667,E2 -12082.667} C_VEL
LIN {X 0,Y 382.985,Z 138.398,A -85,B 0,C 180,E1 -12086.131,E2 -12086.131} C_VEL
LIN {X 0,Y 382.977,Z 138.381,A -85,B 0,C 180,E1 -12089.702,E2 -12089.702} C_VEL
LIN {X 0,Y 383.003,Z 138.402,A -85,B 0,C 180,E1 -12093.401,E2 -12093.401} C_VEL
LIN {X 0,Y 383.025,Z 138.39,A -85,B 0,C 180,E1 -12096.162,E2 -12096.162} C_VEL
LIN {X 0,Y 382.99,Z 138.393,A -85,B 0,C 180,E1 -12099.581,E2 -12099.581} C_VEL
LIN {X 0,Y 383.011,Z 138.402,A -85,B 0,C 180,E1 -12102.779,E2 -12102.779} C_VEL
LIN {X 0,Y 382.994,Z 138.383,A -85,B 0,C 180,E1 -12105.788,E2 -12105.788} C_VEL
LIN {X 0,Y 382.966,Z 138.409,A -85,B 0,C 180,E1 -12108.801,E2 -12108.801} C_VEL
LIN {X 0,Y 382.998,Z 138.391,A -85,B 0,C 180,E1 -12112.098,E2 -12112.098} C_VEL
LIN {X 0,Y 383.022,Z 138.397,A -85,B 0,C 180,E1 -12115.332,E2 -12115.332} C_VEL
LIN {X 0,Y 382.987,Z 138.404,A -85,B 0,C 180,E1 -12119.081,E2 -12119.081} C_VEL
LIN {X 0,Y 382.987,Z 138.406,A -85,B 0,C 180,E1 -12122.692,E2 -12122.692} C_VEL
LIN {X 0,Y 383.015,Z 138.403,A -85,B 0,C 180,E1 -12126.191,E2 -12126.191} C_VEL
LIN {X 0,Y 383.061,Z 138.395,A -85,B 0,C 180,E1 -12129.598,E2 -12129.598} C_VEL
LIN {X 0,Y 383.1,Z 138.376,A -85,B 0,C 180,E1 -12132.931,E2 -12132.931} C_VEL
LIN {X 0,Y 383.131,Z 138.375,A -85,B 0,C 180,E1 -12136.464,E2 -12136.464} C_VEL
LIN {X 0,Y 383.123,Z 138.453,A -85,B 0,C 180,E1 -12138.09,E2 -12138.09} C_VEL
LIN {X 0,Y 384.989,Z 146.23,A -85,B 0,C 180,E1 -12139.856,E2 -12139.856} C_VEL
LIN {X 0,Y 396.473,Z 173.709,A -85,B 0,C 180,E1 -12141.212,E2 -12141.212} C_VEL
LIN {X 0,Y 397.5,Z 177.461,A -85,B 0,C 180,E1 -12141.356,E2 -12141.356} C_VEL
LIN {X 0,Y 394.739,Z 310.552,A -85,B 0,C 180,E1 -12143.835,E2 -12143.835} C_VEL
LIN {X 0,Y 394.013,Z 326.567,A -85,B 0,C 180,E1 -12144.338,E2 -12144.338} C_VEL
LIN {X 0,Y 393.115,Z 341.088,A -85,B 0,C 180,E1 -12145,E2 -12145} C_VEL
LIN {X 0,Y 391.952,Z 355.77,A -85,B 0,C 180,E1 -12145.887,E2 -12145.887} C_VEL
LIN {X 0,Y 390.689,Z 369.088,A -85,B 0,C 180,E1 -12146.906,E2 -12146.906} C_VEL
LIN {X 0,Y 389.241,Z 382.69,A -85,B 0,C 180,E1 -12148.189,E2 -12148.189} C_VEL
LIN {X 0,Y 387.843,Z 395.002,A -85,B 0,C 180,E1 -12149.61,E2 -12149.61} C_VEL
LIN {X 0,Y 386.359,Z 407.112,A -85,B 0,C 180,E1 -12151.302,E2 -12151.302} C_VEL
LIN {X 0,Y 386.296,Z 407.695,A -85,B 0,C 180,E1 -12151.397,E2 -12151.397} C_VEL
LIN {X 0,Y 385.218,Z 411.743,A -85,B 0,C 180,E1 -12152.024,E2 -12152.024} C_VEL
LIN {X 0,Y 381.67,Z 418.04,A -85,B 0,C 180,E1 -12153.031,E2 -12153.031} C_VEL
LIN {X 0,Y 378.102,Z 423.968,A -85,B 0,C 180,E1 -12154.104,E2 -12154.104} C_VEL
LIN {X 0,Y 377.01,Z 427.27,A -85,B 0,C 180,E1 -12154.83,E2 -12154.83} C_VEL
LIN {X 0,Y 376.046,Z 435.604,A -85,B 0,C 180,E1 -12156.977,E2 -12156.977} C_VEL
LIN {X 0,Y 375.312,Z 442.383,A -85,B 0,C 180,E1 -12159.158,E2 -12159.158} C_VEL
LIN {X 0,Y 374.896,Z 447.69,A -85,B 0,C 180,E1 -12161.352,E2 -12161.352} C_VEL
LIN {X 0,Y 374.636,Z 450.758,A -85,B 0,C 180,E1 -12163.009,E2 -12163.009} C_VEL
LIN {X 0,Y 374.385,Z 453.763,A -85,B 0,C 180,E1 -12165.236,E2 -12165.236} C_VEL
LIN {X 0,Y 374.308,Z 455.523,A -85,B 0,C 180,E1 -12167.482,E2 -12167.482} C_VEL
LIN {X 0,Y 374.345,Z 456.046,A -85,B 0,C 180,E1 -12169.751,E2 -12169.751} C_VEL
LIN {X 0,Y 374.375,Z 455.299,A -85,B 0,C 180,E1 -12172.052,E2 -12172.052} C_VEL
LIN {X 0,Y 374.599,Z 453.224,A -85,B 0,C 180,E1 -12174.377,E2 -12174.377} C_VEL
LIN {X 0,Y 375.031,Z 449.727,A -85,B 0,C 180,E1 -12176.728,E2 -12176.728} C_VEL
LIN {X 0,Y 375.591,Z 444.673,A -85,B 0,C 180,E1 -12179.111,E2 -12179.111} C_VEL
LIN {X 0,Y 376.323,Z 439.254,A -85,B 0,C 180,E1 -12181.078,E2 -12181.078} C_VEL
LIN {X 0,Y 377.346,Z 432.504,A -85,B 0,C 180,E1 -12183.057,E2 -12183.057} C_VEL
LIN {X 0,Y 378.657,Z 423.89,A -85,B 0,C 180,E1 -12185.125,E2 -12185.125} C_VEL
LIN {X 0,Y 380.153,Z 414.75,A -85,B 0,C 180,E1 -12186.929,E2 -12186.929} C_VEL
LIN {X 0,Y 381.596,Z 405.764,A -85,B 0,C 180,E1 -12188.432,E2 -12188.432} C_VEL
LIN {X 0,Y 383.466,Z 394.033,A -85,B 0,C 180,E1 -12190.072,E2 -12190.072} C_VEL
LIN {X 0,Y 385.174,Z 382.336,A -85,B 0,C 180,E1 -12191.434,E2 -12191.434} C_VEL
LIN {X 0,Y 386.811,Z 370.374,A -85,B 0,C 180,E1 -12192.594,E2 -12192.594} C_VEL
LIN {X 0,Y 388.391,Z 357.262,A -85,B 0,C 180,E1 -12193.63,E2 -12193.63} C_VEL
LIN {X 0,Y 389.762,Z 343.366,A -85,B 0,C 180,E1 -12194.506,E2 -12194.506} C_VEL
LIN {X 0,Y 390.919,Z 328.243,A -85,B 0,C 180,E1 -12195.233,E2 -12195.233} C_VEL
LIN {X 0,Y 391.884,Z 312.839,A -85,B 0,C 180,E1 -12195.739,E2 -12195.739} C_VEL
LIN {X 0,Y 392.976,Z 272.319,A -85,B 0,C 180,E1 -12196.55,E2 -12196.55} C_VEL
LIN {X 0,Y 395.413,Z 181.596,A -85,B 0,C 180,E1 -12198.286,E2 -12198.286} C_VEL
LIN {X 0,Y 387.36,Z 164.333,A -85,B 0,C 180,E1 -12199.46,E2 -12199.46} C_VEL
LIN {X 0,Y 379.798,Z 150.257,A -85,B 0,C 180,E1 -12200.584,E2 -12200.584} C_VEL
LIN {X 0,Y 378.176,Z 147.044,A -85,B 0,C 180,E1 -12200.855,E2 -12200.855} C_VEL
LIN {X 0,Y 375.958,Z 139.279,A -85,B 0,C 180,E1 -12203.091,E2 -12203.091} C_VEL
LIN {X 0,Y 375.961,Z 139.274,A -85,B 0,C 180,E1 -12205.888,E2 -12205.888} C_VEL
LIN {X 0,Y 375.964,Z 139.279,A -85,B 0,C 180,E1 -12209.687,E2 -12209.687} C_VEL
LIN {X 0,Y 375.965,Z 139.277,A -85,B 0,C 180,E1 -12213.343,E2 -12213.343} C_VEL
LIN {X 0,Y 375.978,Z 139.266,A -85,B 0,C 180,E1 -12216.887,E2 -12216.887} C_VEL
LIN {X 0,Y 375.997,Z 139.275,A -85,B 0,C 180,E1 -12220.339,E2 -12220.339} C_VEL
LIN {X 0,Y 376.026,Z 139.274,A -85,B 0,C 180,E1 -12223.718,E2 -12223.718} C_VEL
LIN {X 0,Y 376.104,Z 139.261,A -85,B 0,C 180,E1 -12227.042,E2 -12227.042} C_VEL
LIN {X 0,Y 376.119,Z 139.256,A -85,B 0,C 180,E1 -12230.318,E2 -12230.318} C_VEL
LIN {X 0,Y 376.23,Z 139.244,A -85,B 0,C 180,E1 -12232.486,E2 -12232.486} C_VEL
LIN {X 0,Y 376.169,Z 139.244,A -85,B 0,C 180,E1 -12234.639,E2 -12234.639} C_VEL
LIN {X 0,Y 376.351,Z 139.223,A -85,B 0,C 180,E1 -12237.859,E2 -12237.859} C_VEL
LIN {X 0,Y 376.487,Z 139.212,A -85,B 0,C 180,E1 -12240,E2 -12240} C_VEL
LIN {X 0,Y 376.184,Z 139.252,A -85,B 0,C 180,E1 -12243.213,E2 -12243.213} C_VEL
LIN {X 0,Y 376.214,Z 139.244,A -85,B 0,C 180,E1 -12246.435,E2 -12246.435} C_VEL
LIN {X 0,Y 376.113,Z 139.258,A -85,B 0,C 180,E1 -12249.681,E2 -12249.681} C_VEL
LIN {X 0,Y 376.088,Z 139.262,A -85,B 0,C 180,E1 -12253.657,E2 -12253.657} C_VEL
LIN {X 0,Y 376.043,Z 139.268,A -85,B 0,C 180,E1 -12257.607,E2 -12257.607} C_VEL
LIN {X 0,Y 375.977,Z 139.276,A -85,B 0,C 180,E1 -12260.832,E2 -12260.832} C_VEL
LIN {X 0,Y 375.993,Z 139.273,A -85,B 0,C 180,E1 -12264.281,E2 -12264.281} C_VEL
LIN {X 0,Y 376.018,Z 139.268,A -85,B 0,C 180,E1 -12266.652,E2 -12266.652} C_VEL
LIN {X 0,Y 375.969,Z 139.272,A -85,B 0,C 180,E1 -12269.079,E2 -12269.079} C_VEL
LIN {X 0,Y 375.947,Z 139.279,A -85,B 0,C 180,E1 -12272.828,E2 -12272.828} C_VEL
LIN {X 0,Y 375.955,Z 139.277,A -85,B 0,C 180,E1 -12275.415,E2 -12275.415} C_VEL
LIN {X 0,Y 375.971,Z 139.262,A -85,B 0,C 180,E1 -12278.27,E2 -12278.27} C_VEL
LIN {X 0,Y 375.932,Z 139.283,A -85,B 0,C 180,E1 -12281.601,E2 -12281.601} C_VEL
LIN {X 0,Y 375.95,Z 139.281,A -85,B 0,C 180,E1 -12285.265,E2 -12285.265} C_VEL
LIN {X 0,Y 375.938,Z 139.278,A -85,B 0,C 180,E1 -12289.133,E2 -12289.133} C_VEL
LIN {X 0,Y 375.956,Z 139.355,A -85,B 0,C 180,E1 -12292.589,E2 -12292.589} C_VEL
LIN {X 0,Y 379.81,Z 152.373,A -85,B 0,C 180,E1 -12295.963,E2 -12295.963} C_VEL
LIN {X 0,Y 382.763,Z 163.905,A -85,B 0,C 180,E1 -12298.712,E2 -12298.712} C_VEL
LIN {X 0,Y 389.412,Z 178,A -85,B 0,C 180,E1 -12299.708,E2 -12299.708} C_VEL
LIN {X 0,Y 393.556,Z 197.911,A -85,B 0,C 180,E1 -12300.55,E2 -12300.55} C_VEL
LIN {X 0,Y 394.93,Z 205.688,A -85,B 0,C 180,E1 -12300.849,E2 -12300.849} C_VEL
LIN {X 0,Y 391.509,Z 331.082,A -85,B 0,C 180,E1 -12303.263,E2 -12303.263} C_VEL
LIN {X 0,Y 390.483,Z 346.762,A -85,B 0,C 180,E1 -12303.764,E2 -12303.764} C_VEL
LIN {X 0,Y 389.368,Z 359.316,A -85,B 0,C 180,E1 -12304.33,E2 -12304.33} C_VEL
LIN {X 0,Y 387.913,Z 373.426,A -85,B 0,C 180,E1 -12305.161,E2 -12305.161} C_VEL
LIN {X 0,Y 386.347,Z 386.379,A -85,B 0,C 180,E1 -12306.125,E2 -12306.125} C_VEL
LIN {X 0,Y 384.322,Z 400.457,A -85,B 0,C 180,E1 -12307.417,E2 -12307.417} C_VEL
LIN {X 0,Y 382.468,Z 413.164,A -85,B 0,C 180,E1 -12308.862,E2 -12308.862} C_VEL
LIN {X 0,Y 380.602,Z 425.048,A -85,B 0,C 180,E1 -12310.497,E2 -12310.497} C_VEL
LIN {X 0,Y 379.033,Z 435.249,A -85,B 0,C 180,E1 -12312.186,E2 -12312.186} C_VEL
LIN {X 0,Y 377.614,Z 444.738,A -85,B 0,C 180,E1 -12314.067,E2 -12314.067} C_VEL
LIN {X 0,Y 376.434,Z 452.671,A -85,B 0,C 180,E1 -12315.954,E2 -12315.954} C_VEL
LIN {X 0,Y 375.607,Z 460.102,A -85,B 0,C 180,E1 -12318.123,E2 -12318.123} C_VEL
LIN {X 0,Y 374.962,Z 466.026,A -85,B 0,C 180,E1 -12320.289,E2 -12320.289} C_VEL
LIN {X 0,Y 374.65,Z 470.605,A -85,B 0,C 180,E1 -12322.455,E2 -12322.455} C_VEL
LIN {X 0,Y 374.488,Z 473.9,A -85,B 0,C 180,E1 -12324.616,E2 -12324.616} C_VEL
LIN {X 0,Y 374.434,Z 475.981,A -85,B 0,C 180,E1 -12326.772,E2 -12326.772} C_VEL
LIN {X 0,Y 374.513,Z 476.917,A -85,B 0,C 180,E1 -12328.925,E2 -12328.925} C_VEL
LIN {X 0,Y 374.514,Z 476.713,A -85,B 0,C 180,E1 -12331.076,E2 -12331.076} C_VEL
LIN {X 0,Y 374.438,Z 475.355,A -85,B 0,C 180,E1 -12333.228,E2 -12333.228} C_VEL
LIN {X 0,Y 374.502,Z 472.772,A -85,B 0,C 180,E1 -12335.385,E2 -12335.385} C_VEL
LIN {X 0,Y 374.648,Z 468.934,A -85,B 0,C 180,E1 -12337.546,E2 -12337.546} C_VEL
LIN {X 0,Y 374.891,Z 463.754,A -85,B 0,C 180,E1 -12339.714,E2 -12339.714} C_VEL
LIN {X 0,Y 375.469,Z 457.102,A -85,B 0,C 180,E1 -12341.883,E2 -12341.883} C_VEL
LIN {X 0,Y 376.017,Z 450.625,A -85,B 0,C 180,E1 -12343.612,E2 -12343.612} C_VEL
LIN {X 0,Y 376.946,Z 442.623,A -85,B 0,C 180,E1 -12345.408,E2 -12345.408} C_VEL
LIN {X 0,Y 378.157,Z 432.454,A -85,B 0,C 180,E1 -12347.299,E2 -12347.299} C_VEL
LIN {X 0,Y 379.507,Z 421.69,A -85,B 0,C 180,E1 -12348.964,E2 -12348.964} C_VEL
LIN {X 0,Y 380.909,Z 409.591,A -85,B 0,C 180,E1 -12350.522,E2 -12350.522} C_VEL
LIN {X 0,Y 382.456,Z 397.099,A -85,B 0,C 180,E1 -12351.847,E2 -12351.847} C_VEL
LIN {X 0,Y 383.933,Z 383.42,A -85,B 0,C 180,E1 -12353.034,E2 -12353.034} C_VEL
LIN {X 0,Y 385.296,Z 369.531,A -85,B 0,C 180,E1 -12353.998,E2 -12353.998} C_VEL
LIN {X 0,Y 386.492,Z 354.713,A -85,B 0,C 180,E1 -12354.795,E2 -12354.795} C_VEL
LIN {X 0,Y 387.497,Z 338.919,A -85,B 0,C 180,E1 -12355.408,E2 -12355.408} C_VEL
LIN {X 0,Y 388.078,Z 323.282,A -85,B 0,C 180,E1 -12355.799,E2 -12355.799} C_VEL
LIN {X 0,Y 390.619,Z 204.315,A -85,B 0,C 180,E1 -12358.027,E2 -12358.027} C_VEL
LIN {X 0,Y 384.38,Z 170.699,A -85,B 0,C 180,E1 -12359.142,E2 -12359.142} C_VEL
LIN {X 0,Y 382.076,Z 164.66,A -85,B 0,C 180,E1 -12359.444,E2 -12359.444} C_VEL
LIN {X 0,Y 378.587,Z 149.68,A -85,B 0,C 180,E1 -12362.572,E2 -12362.572} C_VEL
LIN {X 0,Y 375.985,Z 139.283,A -85,B 0,C 180,E1 -12364.887,E2 -12364.887} C_VEL
LIN {X 0,Y 375.975,Z 139.276,A -85,B 0,C 180,E1 -12368.271,E2 -12368.271} C_VEL
LIN {X 0,Y 375.934,Z 139.284,A -85,B 0,C 180,E1 -12371.601,E2 -12371.601} C_VEL
LIN {X 0,Y 375.928,Z 139.288,A -85,B 0,C 180,E1 -12375.269,E2 -12375.269} C_VEL
LIN {X 0,Y 375.936,Z 139.283,A -85,B 0,C 180,E1 -12378.4,E2 -12378.4} C_VEL
LIN {X 0,Y 375.974,Z 139.273,A -85,B 0,C 180,E1 -12381.731,E2 -12381.731} C_VEL
LIN {X 0,Y 375.982,Z 139.277,A -85,B 0,C 180,E1 -12385.333,E2 -12385.333} C_VEL
LIN {X 0,Y 375.96,Z 139.276,A -85,B 0,C 180,E1 -12388.439,E2 -12388.439} C_VEL
LIN {X 0,Y 375.93,Z 139.261,A -85,B 0,C 180,E1 -12392.136,E2 -12392.136} C_VEL
LIN {X 0,Y 375.978,Z 139.273,A -85,B 0,C 180,E1 -12395.718,E2 -12395.718} C_VEL
LIN {X 0,Y 376.002,Z 139.272,A -85,B 0,C 180,E1 -12399.199,E2 -12399.199} C_VEL
LIN {X 0,Y 376.036,Z 139.265,A -85,B 0,C 180,E1 -12402.601,E2 -12402.601} C_VEL
LIN {X 0,Y 376.094,Z 139.263,A -85,B 0,C 180,E1 -12406.343,E2 -12406.343} C_VEL
LIN {X 0,Y 376.117,Z 139.261,A -85,B 0,C 180,E1 -12410.319,E2 -12410.319} C_VEL
LIN {X 0,Y 376.202,Z 139.244,A -85,B 0,C 180,E1 -12413.565,E2 -12413.565} C_VEL
LIN {X 0,Y 376.342,Z 139.217,A -85,B 0,C 180,E1 -12417.86,E2 -12417.86} C_VEL
LIN {X 0,Y 376.337,Z 139.222,A -85,B 0,C 180,E1 -12422.141,E2 -12422.141} C_VEL
LIN {X 0,Y 376.197,Z 139.24,A -85,B 0,C 180,E1 -12426.444,E2 -12426.444} C_VEL
LIN {X 0,Y 376.111,Z 139.232,A -85,B 0,C 180,E1 -12429.682,E2 -12429.682} C_VEL
LIN {X 0,Y 376.045,Z 139.266,A -85,B 0,C 180,E1 -12433.626,E2 -12433.626} C_VEL
LIN {X 0,Y 375.984,Z 139.271,A -85,B 0,C 180,E1 -12437.576,E2 -12437.576} C_VEL
LIN {X 0,Y 375.951,Z 139.277,A -85,B 0,C 180,E1 -12440.819,E2 -12440.819} C_VEL
LIN {X 0,Y 375.938,Z 139.279,A -85,B 0,C 180,E1 -12444.286,E2 -12444.286} C_VEL
LIN {X 0,Y 375.914,Z 139.279,A -85,B 0,C 180,E1 -12446.661,E2 -12446.661} C_VEL
LIN {X 0,Y 375.917,Z 139.26,A -85,B 0,C 180,E1 -12449.084,E2 -12449.084} C_VEL
LIN {X 0,Y 375.957,Z 139.27,A -85,B 0,C 180,E1 -12451.563,E2 -12451.563} C_VEL
LIN {X 0,Y 375.953,Z 139.274,A -85,B 0,C 180,E1 -12455.417,E2 -12455.417} C_VEL
LIN {X 0,Y 375.938,Z 139.258,A -85,B 0,C 180,E1 -12458.263,E2 -12458.263} C_VEL
LIN {X 0,Y 375.922,Z 139.281,A -85,B 0,C 180,E1 -12461.598,E2 -12461.598} C_VEL
LIN {X 0,Y 375.925,Z 139.271,A -85,B 0,C 180,E1 -12464.73,E2 -12464.73} C_VEL
LIN {X 0,Y 375.93,Z 139.277,A -85,B 0,C 180,E1 -12467.699,E2 -12467.699} C_VEL
LIN {X 0,Y 375.939,Z 139.279,A -85,B 0,C 180,E1 -12470.534,E2 -12470.534} C_VEL
LIN {X 0,Y 375.967,Z 139.272,A -85,B 0,C 180,E1 -12473.496,E2 -12473.496} C_VEL
LIN {X 0,Y 375.964,Z 139.277,A -85,B 0,C 180,E1 -12475.888,E2 -12475.888} C_VEL
LIN {X 0,Y 375.967,Z 139.279,A -85,B 0,C 180,E1 -12479.687,E2 -12479.687} C_VEL
LIN {X 0,Y 375.93,Z 139.279,A -85,B 0,C 180,E1 -12482.135,E2 -12482.135} C_VEL
LIN {X 0,Y 375.964,Z 139.282,A -85,B 0,C 180,E1 -12485.716,E2 -12485.716} C_VEL
LIN {X 0,Y 376.004,Z 139.272,A -85,B 0,C 180,E1 -12489.198,E2 -12489.198} C_VEL
LIN {X 0,Y 376.038,Z 139.253,A -85,B 0,C 180,E1 -12492.6,E2 -12492.6} C_VEL
LIN {X 0,Y 376.095,Z 139.251,A -85,B 0,C 180,E1 -12496.342,E2 -12496.342} C_VEL
LIN {X 0,Y 376.114,Z 139.364,A -85,B 0,C 180,E1 -12497.693,E2 -12497.693} C_VEL
LIN {X 0,Y 377.794,Z 146.455,A -85,B 0,C 180,E1 -12499.331,E2 -12499.331} C_VEL
LIN {X 0,Y 387.439,Z 169.224,A -85,B 0,C 180,E1 -12500.503,E2 -12500.503} C_VEL
LIN {X 0,Y 390.986,Z 178.209,A -85,B 0,C 180,E1 -12500.93,E2 -12500.93} C_VEL
LIN {X 0,Y 388.986,Z 274.165,A -85,B 0,C 180,E1 -12502.734,E2 -12502.734} C_VEL
LIN {X 0,Y 388.129,Z 311.765,A -85,B 0,C 180,E1 -12503.469,E2 -12503.469} C_VEL
LIN {X 0,Y 387.383,Z 327.384,A -85,B 0,C 180,E1 -12503.979,E2 -12503.979} C_VEL
LIN {X 0,Y 386.455,Z 341.775,A -85,B 0,C 180,E1 -12504.652,E2 -12504.652} C_VEL
LIN {X 0,Y 385.275,Z 356.33,A -85,B 0,C 180,E1 -12505.553,E2 -12505.553} C_VEL
LIN {X 0,Y 383.954,Z 369.602,A -85,B 0,C 180,E1 -12506.589,E2 -12506.589} C_VEL
LIN {X 0,Y 382.463,Z 383.138,A -85,B 0,C 180,E1 -12507.893,E2 -12507.893} C_VEL
LIN {X 0,Y 380.979,Z 395.423,A -85,B 0,C 180,E1 -12509.339,E2 -12509.339} C_VEL
LIN {X 0,Y 379.568,Z 406.727,A -85,B 0,C 180,E1 -12510.944,E2 -12510.944} C_VEL
LIN {X 0,Y 378.288,Z 416.814,A -85,B 0,C 180,E1 -12512.662,E2 -12512.662} C_VEL
LIN {X 0,Y 377.129,Z 426.004,A -85,B 0,C 180,E1 -12514.542,E2 -12514.542} C_VEL
LIN {X 0,Y 377.01,Z 427.27,A -85,B 0,C 180,E1 -12514.83,E2 -12514.83} C_VEL
LIN {X 0,Y 375.961,Z 430.463,A -85,B 0,C 180,E1 -12515.576,E2 -12515.576} C_VEL
LIN {X 0,Y 372.567,Z 435.354,A -85,B 0,C 180,E1 -12516.788,E2 -12516.788} C_VEL
LIN {X 0,Y 369.243,Z 439.815,A -85,B 0,C 180,E1 -12518.058,E2 -12518.058} C_VEL
LIN {X 0,Y 368.319,Z 442.201,A -85,B 0,C 180,E1 -12518.887,E2 -12518.887} C_VEL
LIN {X 0,Y 367.869,Z 447.371,A -85,B 0,C 180,E1 -12521.013,E2 -12521.013} C_VEL
LIN {X 0,Y 367.494,Z 451.467,A -85,B 0,C 180,E1 -12523.267,E2 -12523.267} C_VEL
LIN {X 0,Y 367.276,Z 454.286,A -85,B 0,C 180,E1 -12525.539,E2 -12525.539} C_VEL
LIN {X 0,Y 367.211,Z 455.865,A -85,B 0,C 180,E1 -12527.831,E2 -12527.831} C_VEL
LIN {X 0,Y 367.253,Z 456.179,A -85,B 0,C 180,E1 -12530.33,E2 -12530.33} C_VEL
LIN {X 0,Y 367.315,Z 455.267,A -85,B 0,C 180,E1 -12532.499,E2 -12532.499} C_VEL
LIN {X 0,Y 367.573,Z 452.993,A -85,B 0,C 180,E1 -12534.875,E2 -12534.875} C_VEL
LIN {X 0,Y 367.845,Z 451.269,A -85,B 0,C 180,E1 -12536.105,E2 -12536.105} C_VEL
LIN {X 0,Y 368.318,Z 446.849,A -85,B 0,C 180,E1 -12538.491,E2 -12538.491} C_VEL
LIN {X 0,Y 369.177,Z 440.723,A -85,B 0,C 180,E1 -12540.93,E2 -12540.93} C_VEL
LIN {X 0,Y 370.305,Z 433.85,A -85,B 0,C 180,E1 -12543.068,E2 -12543.068} C_VEL
LIN {X 0,Y 371.682,Z 425.305,A -85,B 0,C 180,E1 -12545.219,E2 -12545.219} C_VEL
LIN {X 0,Y 373.22,Z 416.436,A -85,B 0,C 180,E1 -12547.055,E2 -12547.055} C_VEL
LIN {X 0,Y 375.036,Z 405.777,A -85,B 0,C 180,E1 -12548.886,E2 -12548.886} C_VEL
LIN {X 0,Y 376.922,Z 394.55,A -85,B 0,C 180,E1 -12550.482,E2 -12550.482} C_VEL
LIN {X 0,Y 378.756,Z 382.476,A -85,B 0,C 180,E1 -12551.912,E2 -12551.912} C_VEL
LIN {X 0,Y 380.531,Z 370.265,A -85,B 0,C 180,E1 -12553.106,E2 -12553.106} C_VEL
LIN {X 0,Y 382.218,Z 356.738,A -85,B 0,C 180,E1 -12554.183,E2 -12554.183} C_VEL
LIN {X 0,Y 383.728,Z 341.829,A -85,B 0,C 180,E1 -12555.118,E2 -12555.118} C_VEL
LIN {X 0,Y 384.966,Z 326.75,A -85,B 0,C 180,E1 -12555.821,E2 -12555.821} C_VEL
LIN {X 0,Y 385.839,Z 311.232,A -85,B 0,C 180,E1 -12556.321,E2 -12556.321} C_VEL
LIN {X 0,Y 389.512,Z 183.795,A -85,B 0,C 180,E1 -12558.808,E2 -12558.808} C_VEL
LIN {X 0,Y 381.156,Z 166.088,A -85,B 0,C 180,E1 -12560.066,E2 -12560.066} C_VEL
LIN {X 0,Y 372.857,Z 150.809,A -85,B 0,C 180,E1 -12561.354,E2 -12561.354} C_VEL
LIN {X 0,Y 370.956,Z 147.25,A -85,B 0,C 180,E1 -12561.692,E2 -12561.692} C_VEL
LIN {X 0,Y 368.918,Z 140.161,A -85,B 0,C 180,E1 -12563.803,E2 -12563.803} C_VEL
LIN {X 0,Y 368.898,Z 140.157,A -85,B 0,C 180,E1 -12566.956,E2 -12566.956} C_VEL
LIN {X 0,Y 368.901,Z 140.157,A -85,B 0,C 180,E1 -12570.308,E2 -12570.308} C_VEL
LIN {X 0,Y 368.959,Z 140.153,A -85,B 0,C 180,E1 -12574.016,E2 -12574.016} C_VEL
LIN {X 0,Y 368.922,Z 140.151,A -85,B 0,C 180,E1 -12577.604,E2 -12577.604} C_VEL
LIN {X 0,Y 368.955,Z 140.152,A -85,B 0,C 180,E1 -12581.105,E2 -12581.105} C_VEL
LIN {X 0,Y 368.997,Z 140.142,A -85,B 0,C 180,E1 -12584.535,E2 -12584.535} C_VEL
LIN {X 0,Y 369.005,Z 140.14,A -85,B 0,C 180,E1 -12587.906,E2 -12587.906} C_VEL
LIN {X 0,Y 369.229,Z 140.114,A -85,B 0,C 180,E1 -12591.8,E2 -12591.8} C_VEL
LIN {X 0,Y 369.143,Z 140.12,A -85,B 0,C 180,E1 -12594.537,E2 -12594.537} C_VEL
LIN {X 0,Y 369.316,Z 140.1,A -85,B 0,C 180,E1 -12597.818,E2 -12597.818} C_VEL
LIN {X 0,Y 369.457,Z 140.088,A -85,B 0,C 180,E1 -12600,E2 -12600} C_VEL
LIN {X 0,Y 369.316,Z 140.102,A -85,B 0,C 180,E1 -12602.181,E2 -12602.181} C_VEL
LIN {X 0,Y 369.173,Z 140.122,A -85,B 0,C 180,E1 -12606.558,E2 -12606.558} C_VEL
LIN {X 0,Y 369.063,Z 140.136,A -85,B 0,C 180,E1 -12609.868,E2 -12609.868} C_VEL
LIN {X 0,Y 369.036,Z 140.14,A -85,B 0,C 180,E1 -12613.772,E2 -12613.772} C_VEL
LIN {X 0,Y 369,Z 140.145,A -85,B 0,C 180,E1 -12617.768,E2 -12617.768} C_VEL
LIN {X 0,Y 368.928,Z 140.156,A -85,B 0,C 180,E1 -12621.219,E2 -12621.219} C_VEL
LIN {X 0,Y 368.956,Z 140.154,A -85,B 0,C 180,E1 -12624.775,E2 -12624.775} C_VEL
LIN {X 0,Y 368.967,Z 140.151,A -85,B 0,C 180,E1 -12627.203,E2 -12627.203} C_VEL
LIN {X 0,Y 368.917,Z 140.151,A -85,B 0,C 180,E1 -12629.69,E2 -12629.69} C_VEL
LIN {X 0,Y 368.895,Z 140.159,A -85,B 0,C 180,E1 -12633.043,E2 -12633.043} C_VEL
LIN {X 0,Y 368.915,Z 140.158,A -85,B 0,C 180,E1 -12636.197,E2 -12636.197} C_VEL
LIN {X 0,Y 368.899,Z 140.141,A -85,B 0,C 180,E1 -12638.953,E2 -12638.953} C_VEL
LIN {X 0,Y 368.879,Z 140.154,A -85,B 0,C 180,E1 -12642.009,E2 -12642.009} C_VEL
LIN {X 0,Y 368.904,Z 140.159,A -85,B 0,C 180,E1 -12645.18,E2 -12645.18} C_VEL
LIN {X 0,Y 368.881,Z 140.161,A -85,B 0,C 180,E1 -12648.178,E2 -12648.178} C_VEL
LIN {X 0,Y 368.964,Z 140.33,A -85,B 0,C 180,E1 -12651.883,E2 -12651.883} C_VEL
LIN {X 0,Y 372.727,Z 152.966,A -85,B 0,C 180,E1 -12655.281,E2 -12655.281} C_VEL
LIN {X 0,Y 375.6,Z 163.807,A -85,B 0,C 180,E1 -12657.927,E2 -12657.927} C_VEL
LIN {X 0,Y 383.602,Z 180.49,A -85,B 0,C 180,E1 -12659.179,E2 -12659.179} C_VEL
LIN {X 0,Y 386.56,Z 193.542,A -85,B 0,C 180,E1 -12659.773,E2 -12659.773} C_VEL
LIN {X 0,Y 388.936,Z 207.466,A -85,B 0,C 180,E1 -12660.317,E2 -12660.317} C_VEL
LIN {X 0,Y 385.404,Z 330.845,A -85,B 0,C 180,E1 -12662.732,E2 -12662.732} C_VEL
LIN {X 0,Y 384.33,Z 346.512,A -85,B 0,C 180,E1 -12663.237,E2 -12663.237} C_VEL
LIN {X 0,Y 383.043,Z 360.348,A -85,B 0,C 180,E1 -12663.874,E2 -12663.874} C_VEL
LIN {X 0,Y 381.356,Z 375.682,A -85,B 0,C 180,E1 -12664.818,E2 -12664.818} C_VEL
LIN {X 0,Y 379.49,Z 390.02,A -85,B 0,C 180,E1 -12665.957,E2 -12665.957} C_VEL
LIN {X 0,Y 377.454,Z 403.386,A -85,B 0,C 180,E1 -12667.273,E2 -12667.273} C_VEL
LIN {X 0,Y 375.526,Z 415.581,A -85,B 0,C 180,E1 -12668.74,E2 -12668.74} C_VEL
LIN {X 0,Y 373.526,Z 427.564,A -85,B 0,C 180,E1 -12670.49,E2 -12670.49} C_VEL
LIN {X 0,Y 371.99,Z 436.872,A -85,B 0,C 180,E1 -12672.121,E2 -12672.121} C_VEL
LIN {X 0,Y 370.535,Z 446.038,A -85,B 0,C 180,E1 -12674.037,E2 -12674.037} C_VEL
LIN {X 0,Y 369.169,Z 454.383,A -85,B 0,C 180,E1 -12676.144,E2 -12676.144} C_VEL
LIN {X 0,Y 368.609,Z 460.071,A -85,B 0,C 180,E1 -12677.894,E2 -12677.894} C_VEL
LIN {X 0,Y 367.907,Z 465.956,A -85,B 0,C 180,E1 -12680.101,E2 -12680.101} C_VEL
LIN {X 0,Y 367.574,Z 470.499,A -85,B 0,C 180,E1 -12682.309,E2 -12682.309} C_VEL
LIN {X 0,Y 367.41,Z 473.777,A -85,B 0,C 180,E1 -12684.512,E2 -12684.512} C_VEL
LIN {X 0,Y 367.351,Z 475.823,A -85,B 0,C 180,E1 -12686.71,E2 -12686.71} C_VEL
LIN {X 0,Y 367.412,Z 476.725,A -85,B 0,C 180,E1 -12688.904,E2 -12688.904} C_VEL
LIN {X 0,Y 367.414,Z 476.489,A -85,B 0,C 180,E1 -12691.096,E2 -12691.096} C_VEL
LIN {X 0,Y 367.354,Z 475.099,A -85,B 0,C 180,E1 -12693.291,E2 -12693.291} C_VEL
LIN {X 0,Y 367.422,Z 472.498,A -85,B 0,C 180,E1 -12695.489,E2 -12695.489} C_VEL
LIN {X 0,Y 367.568,Z 468.62,A -85,B 0,C 180,E1 -12697.692,E2 -12697.692} C_VEL
LIN {X 0,Y 367.817,Z 463.396,A -85,B 0,C 180,E1 -12699.903,E2 -12699.903} C_VEL
LIN {X 0,Y 368.428,Z 456.697,A -85,B 0,C 180,E1 -12702.113,E2 -12702.113} C_VEL
LIN {X 0,Y 369.259,Z 448.32,A -85,B 0,C 180,E1 -12704.326,E2 -12704.326} C_VEL
LIN {X 0,Y 370.308,Z 439.362,A -85,B 0,C 180,E1 -12706.257,E2 -12706.257} C_VEL
LIN {X 0,Y 371.524,Z 430.232,A -85,B 0,C 180,E1 -12707.903,E2 -12707.903} C_VEL
LIN {X 0,Y 372.908,Z 419.366,A -85,B 0,C 180,E1 -12709.555,E2 -12709.555} C_VEL
LIN {X 0,Y 374.37,Z 407.669,A -85,B 0,C 180,E1 -12711.041,E2 -12711.041} C_VEL
LIN {X 0,Y 375.947,Z 394.814,A -85,B 0,C 180,E1 -12712.39,E2 -12712.39} C_VEL
LIN {X 0,Y 377.356,Z 382.432,A -85,B 0,C 180,E1 -12713.46,E2 -12713.46} C_VEL
LIN {X 0,Y 378.818,Z 367.905,A -85,B 0,C 180,E1 -12714.464,E2 -12714.464} C_VEL
LIN {X 0,Y 379.957,Z 353.2,A -85,B 0,C 180,E1 -12715.251,E2 -12715.251} C_VEL
LIN {X 0,Y 381.008,Z 337.815,A -85,B 0,C 180,E1 -12715.836,E2 -12715.836} C_VEL
LIN {X 0,Y 381.563,Z 321.583,A -85,B 0,C 180,E1 -12716.236,E2 -12716.236} C_VEL
LIN {X 0,Y 384.199,Z 206.213,A -85,B 0,C 180,E1 -12718.424,E2 -12718.424} C_VEL
LIN {X 0,Y 378.348,Z 173.581,A -85,B 0,C 180,E1 -12719.517,E2 -12719.517} C_VEL
LIN {X 0,Y 374.776,Z 164.418,A -85,B 0,C 180,E1 -12719.993,E2 -12719.993} C_VEL
LIN {X 0,Y 371.578,Z 150.594,A -85,B 0,C 180,E1 -12722.941,E2 -12722.941} C_VEL
LIN {X 0,Y 368.937,Z 140.161,A -85,B 0,C 180,E1 -12725.306,E2 -12725.306} C_VEL
LIN {X 0,Y 368.903,Z 140.158,A -85,B 0,C 180,E1 -12728.954,E2 -12728.954} C_VEL
LIN {X 0,Y 368.882,Z 140.163,A -85,B 0,C 180,E1 -12732.01,E2 -12732.01} C_VEL
LIN {X 0,Y 368.881,Z 140.165,A -85,B 0,C 180,E1 -12735.176,E2 -12735.176} C_VEL
LIN {X 0,Y 368.885,Z 140.162,A -85,B 0,C 180,E1 -12738.178,E2 -12738.178} C_VEL
LIN {X 0,Y 368.908,Z 140.15,A -85,B 0,C 180,E1 -12741.361,E2 -12741.361} C_VEL
LIN {X 0,Y 368.939,Z 140.153,A -85,B 0,C 180,E1 -12745.147,E2 -12745.147} C_VEL
LIN {X 0,Y 368.932,Z 140.156,A -85,B 0,C 180,E1 -12749.047,E2 -12749.047} C_VEL
LIN {X 0,Y 368.869,Z 140.14,A -85,B 0,C 180,E1 -12752.789,E2 -12752.789} C_VEL
LIN {X 0,Y 368.958,Z 140.149,A -85,B 0,C 180,E1 -12756.421,E2 -12756.421} C_VEL
LIN {X 0,Y 368.939,Z 140.15,A -85,B 0,C 180,E1 -12759.948,E2 -12759.948} C_VEL
LIN {X 0,Y 368.972,Z 140.143,A -85,B 0,C 180,E1 -12763.399,E2 -12763.399} C_VEL
LIN {X 0,Y 369.062,Z 140.135,A -85,B 0,C 180,E1 -12766.791,E2 -12766.791} C_VEL
LIN {X 0,Y 369.067,Z 140.137,A -85,B 0,C 180,E1 -12770.132,E2 -12770.132} C_VEL
LIN {X 0,Y 369.163,Z 140.121,A -85,B 0,C 180,E1 -12773.441,E2 -12773.441} C_VEL
LIN {X 0,Y 369.306,Z 140.094,A -85,B 0,C 180,E1 -12777.819,E2 -12777.819} C_VEL
LIN {X 0,Y 369.3,Z 140.099,A -85,B 0,C 180,E1 -12782.182,E2 -12782.182} C_VEL
LIN {X 0,Y 369.16,Z 140.116,A -85,B 0,C 180,E1 -12786.56,E2 -12786.56} C_VEL
LIN {X 0,Y 369.061,Z 140.11,A -85,B 0,C 180,E1 -12789.869,E2 -12789.869} C_VEL
LIN {X 0,Y 369.006,Z 140.144,A -85,B 0,C 180,E1 -12793.749,E2 -12793.749} C_VEL
LIN {X 0,Y 368.941,Z 140.149,A -85,B 0,C 180,E1 -12797.746,E2 -12797.746} C_VEL
LIN {X 0,Y 368.884,Z 140.159,A -85,B 0,C 180,E1 -12801.223,E2 -12801.223} C_VEL
LIN {X 0,Y 368.912,Z 140.157,A -85,B 0,C 180,E1 -12803.873,E2 -12803.873} C_VEL
LIN {X 0,Y 368.861,Z 140.152,A -85,B 0,C 180,E1 -12807.212,E2 -12807.212} C_VEL
LIN {X 0,Y 368.896,Z 140.133,A -85,B 0,C 180,E1 -12809.693,E2 -12809.693} C_VEL
LIN {X 0,Y 368.9,Z 140.156,A -85,B 0,C 180,E1 -12813.043,E2 -12813.043} C_VEL
LIN {X 0,Y 368.915,Z 140.148,A -85,B 0,C 180,E1 -12816.198,E2 -12816.198} C_VEL
LIN {X 0,Y 368.878,Z 140.14,A -85,B 0,C 180,E1 -12818.957,E2 -12818.957} C_VEL
LIN {X 0,Y 368.875,Z 140.158,A -85,B 0,C 180,E1 -12822.007,E2 -12822.007} C_VEL
LIN {X 0,Y 368.877,Z 140.143,A -85,B 0,C 180,E1 -12825.175,E2 -12825.175} C_VEL
LIN {X 0,Y 368.874,Z 140.157,A -85,B 0,C 180,E1 -12828.176,E2 -12828.176} C_VEL
LIN {X 0,Y 368.881,Z 140.15,A -85,B 0,C 180,E1 -12831.366,E2 -12831.366} C_VEL
LIN {X 0,Y 368.941,Z 140.152,A -85,B 0,C 180,E1 -12835.146,E2 -12835.146} C_VEL
LIN {X 0,Y 368.935,Z 140.155,A -85,B 0,C 180,E1 -12839.046,E2 -12839.046} C_VEL
LIN {X 0,Y 368.87,Z 140.165,A -85,B 0,C 180,E1 -12842.789,E2 -12842.789} C_VEL
LIN {X 0,Y 368.951,Z 140.155,A -85,B 0,C 180,E1 -12846.42,E2 -12846.42} C_VEL
LIN {X 0,Y 368.942,Z 140.156,A -85,B 0,C 180,E1 -12849.947,E2 -12849.947} C_VEL
LIN {X 0,Y 368.974,Z 140.14,A -85,B 0,C 180,E1 -12853.398,E2 -12853.398} C_VEL
LIN {X 0,Y 369.088,Z 140.245,A -85,B 0,C 180,E1 -12857.281,E2 -12857.281} C_VEL
LIN {X 0,Y 370.616,Z 146.689,A -85,B 0,C 180,E1 -12858.787,E2 -12858.787} C_VEL
LIN {X 0,Y 381.247,Z 171.612,A -85,B 0,C 180,E1 -12860.114,E2 -12860.114} C_VEL
LIN {X 0,Y 384.631,Z 180.278,A -85,B 0,C 180,E1 -12860.534,E2 -12860.534} C_VEL
LIN {X 0,Y 381.61,Z 311.618,A -85,B 0,C 180,E1 -12863.058,E2 -12863.058} C_VEL
LIN {X 0,Y 380.821,Z 327.38,A -85,B 0,C 180,E1 -12863.576,E2 -12863.576} C_VEL
LIN {X 0,Y 379.82,Z 342.395,A -85,B 0,C 180,E1 -12864.292,E2 -12864.292} C_VEL
LIN {X 0,Y 378.593,Z 356.876,A -85,B 0,C 180,E1 -12865.208,E2 -12865.208} C_VEL
LIN {X 0,Y 377.217,Z 370.115,A -85,B 0,C 180,E1 -12866.261,E2 -12866.261} C_VEL
LIN {X 0,Y 375.686,Z 383.583,A -85,B 0,C 180,E1 -12867.587,E2 -12867.587} C_VEL
LIN {X 0,Y 374.131,Z 395.837,A -85,B 0,C 180,E1 -12869.058,E2 -12869.058} C_VEL
LIN {X 0,Y 372.528,Z 408.045,A -85,B 0,C 180,E1 -12870.843,E2 -12870.843} C_VEL
LIN {X 0,Y 371.336,Z 417.17,A -85,B 0,C 180,E1 -12872.44,E2 -12872.44} C_VEL
LIN {X 0,Y 370.156,Z 426.328,A -85,B 0,C 180,E1 -12874.355,E2 -12874.355} C_VEL
LIN {X 0,Y 369.186,Z 433.962,A -85,B 0,C 180,E1 -12876.284,E2 -12876.284} C_VEL
LIN {X 0,Y 368.557,Z 440.279,A -85,B 0,C 180,E1 -12878.222,E2 -12878.222} C_VEL
LIN {X 0,Y 368.319,Z 442.201,A -85,B 0,C 180,E1 -12878.887,E2 -12878.887} C_VEL
LIN {X 0,Y 367.434,Z 444.452,A -85,B 0,C 180,E1 -12879.732,E2 -12879.732} C_VEL
LIN {X 0,Y 364.293,Z 447.782,A -85,B 0,C 180,E1 -12881.113,E2 -12881.113} C_VEL
LIN {X 0,Y 361.687,Z 450.064,A -85,B 0,C 180,E1 -12882.246,E2 -12882.246} C_VEL
LIN {X 0,Y 360.5,Z 451.538,A -85,B 0,C 180,E1 -12883.137,E2 -12883.137} C_VEL
LIN {X 0,Y 360.363,Z 452,A -85,B 0,C 180,E1 -12883.441,E2 -12883.441} C_VEL
LIN {X 0,Y 360.184,Z 454.807,A -85,B 0,C 180,E1 -12885.853,E2 -12885.853} C_VEL
LIN {X 0,Y 360.1,Z 456.208,A -85,B 0,C 180,E1 -12888.196,E2 -12888.196} C_VEL
LIN {X 0,Y 360.15,Z 456.361,A -85,B 0,C 180,E1 -12890.564,E2 -12890.564} C_VEL
LIN {X 0,Y 360.253,Z 455.235,A -85,B 0,C 180,E1 -12892.965,E2 -12892.965} C_VEL
LIN {X 0,Y 360.584,Z 452.763,A -85,B 0,C 180,E1 -12895.391,E2 -12895.391} C_VEL
LIN {X 0,Y 361.087,Z 448.846,A -85,B 0,C 180,E1 -12897.847,E2 -12897.847} C_VEL
LIN {X 0,Y 361.871,Z 443.351,A -85,B 0,C 180,E1 -12900.328,E2 -12900.328} C_VEL
LIN {X 0,Y 362.756,Z 438.078,A -85,B 0,C 180,E1 -12902.193,E2 -12902.193} C_VEL
LIN {X 0,Y 364.059,Z 430.501,A -85,B 0,C 180,E1 -12904.378,E2 -12904.378} C_VEL
LIN {X 0,Y 365.521,Z 422.515,A -85,B 0,C 180,E1 -12906.271,E2 -12906.271} C_VEL
LIN {X 0,Y 367.121,Z 413.429,A -85,B 0,C 180,E1 -12908.073,E2 -12908.073} C_VEL
LIN {X 0,Y 369.028,Z 402.82,A -85,B 0,C 180,E1 -12909.819,E2 -12909.819} C_VEL
LIN {X 0,Y 371.139,Z 390.406,A -85,B 0,C 180,E1 -12911.511,E2 -12911.511} C_VEL
LIN {X 0,Y 373.097,Z 378.145,A -85,B 0,C 180,E1 -12912.881,E2 -12912.881} C_VEL
LIN {X 0,Y 375.124,Z 363.969,A -85,B 0,C 180,E1 -12914.17,E2 -12914.17} C_VEL
LIN {X 0,Y 376.849,Z 349.35,A -85,B 0,C 180,E1 -12915.222,E2 -12915.222} C_VEL
LIN {X 0,Y 378.267,Z 334.303,A -85,B 0,C 180,E1 -12916.05,E2 -12916.05} C_VEL
LIN {X 0,Y 379.419,Z 318.817,A -85,B 0,C 180,E1 -12916.658,E2 -12916.658} C_VEL
LIN {X 0,Y 380.075,Z 303.227,A -85,B 0,C 180,E1 -12917.057,E2 -12917.057} C_VEL
LIN {X 0,Y 383.482,Z 185.797,A -85,B 0,C 180,E1 -12919.369,E2 -12919.369} C_VEL
LIN {X 0,Y 375.992,Z 169.882,A -85,B 0,C 180,E1 -12920.54,E2 -12920.54} C_VEL
LIN {X 0,Y 368.35,Z 155.645,A -85,B 0,C 180,E1 -12921.764,E2 -12921.764} C_VEL
LIN {X 0,Y 363.766,Z 147.609,A -85,B 0,C 180,E1 -12922.531,E2 -12922.531} C_VEL
LIN {X 0,Y 361.872,Z 141.028,A -85,B 0,C 180,E1 -12924.557,E2 -12924.557} C_VEL
LIN {X 0,Y 361.849,Z 141.033,A -85,B 0,C 180,E1 -12927.055,E2 -12927.055} C_VEL
LIN {X 0,Y 361.866,Z 141.025,A -85,B 0,C 180,E1 -12930.952,E2 -12930.952} C_VEL
LIN {X 0,Y 361.902,Z 141.024,A -85,B 0,C 180,E1 -12934.707,E2 -12934.707} C_VEL
LIN {X 0,Y 361.88,Z 141.034,A -85,B 0,C 180,E1 -12938.346,E2 -12938.346} C_VEL
LIN {X 0,Y 361.92,Z 141.024,A -85,B 0,C 180,E1 -12942.084,E2 -12942.084} C_VEL
LIN {X 0,Y 361.962,Z 141.018,A -85,B 0,C 180,E1 -12945.379,E2 -12945.379} C_VEL
LIN {X 0,Y 361.971,Z 141.018,A -85,B 0,C 180,E1 -12948.804,E2 -12948.804} C_VEL
LIN {X 0,Y 362.151,Z 140.999,A -85,B 0,C 180,E1 -12952.192,E2 -12952.192} C_VEL
LIN {X 0,Y 362.116,Z 140.995,A -85,B 0,C 180,E1 -12954.431,E2 -12954.431} C_VEL
LIN {X 0,Y 362.28,Z 140.976,A -85,B 0,C 180,E1 -12957.776,E2 -12957.776} C_VEL
LIN {X 0,Y 362.426,Z 140.964,A -85,B 0,C 180,E1 -12960,E2 -12960} C_VEL
LIN {X 0,Y 362.28,Z 140.978,A -85,B 0,C 180,E1 -12962.223,E2 -12962.223} C_VEL
LIN {X 0,Y 362.135,Z 140.999,A -85,B 0,C 180,E1 -12966.686,E2 -12966.686} C_VEL
LIN {X 0,Y 361.999,Z 141.016,A -85,B 0,C 180,E1 -12970.062,E2 -12970.062} C_VEL
LIN {X 0,Y 361.997,Z 141.017,A -85,B 0,C 180,E1 -12973.899,E2 -12973.899} C_VEL
LIN {X 0,Y 361.966,Z 141.021,A -85,B 0,C 180,E1 -12977.938,E2 -12977.938} C_VEL
LIN {X 0,Y 361.891,Z 141.03,A -85,B 0,C 180,E1 -12981.653,E2 -12981.653} C_VEL
LIN {X 0,Y 361.927,Z 141.024,A -85,B 0,C 180,E1 -12985.29,E2 -12985.29} C_VEL
LIN {X 0,Y 361.917,Z 141.028,A -85,B 0,C 180,E1 -12987.778,E2 -12987.778} C_VEL
LIN {X 0,Y 361.845,Z 141.035,A -85,B 0,C 180,E1 -12991.285,E2 -12991.285} C_VEL
LIN {X 0,Y 361.852,Z 141.036,A -85,B 0,C 180,E1 -12994.28,E2 -12994.28} C_VEL
LIN {X 0,Y 361.861,Z 141.031,A -85,B 0,C 180,E1 -12997.223,E2 -12997.223} C_VEL
LIN {X 0,Y 361.834,Z 141.042,A -85,B 0,C 180,E1 -13000.755,E2 -13000.755} C_VEL
LIN {X 0,Y 361.831,Z 141.033,A -85,B 0,C 180,E1 -13004.366,E2 -13004.366} C_VEL
LIN {X 0,Y 361.834,Z 141.03,A -85,B 0,C 180,E1 -13007.568,E2 -13007.568} C_VEL
LIN {X 0,Y 361.87,Z 141.072,A -85,B 0,C 180,E1 -13011.068,E2 -13011.068} C_VEL
LIN {X 0,Y 364.981,Z 151.396,A -85,B 0,C 180,E1 -13013.973,E2 -13013.973} C_VEL
LIN {X 0,Y 367.765,Z 161.442,A -85,B 0,C 180,E1 -13016.593,E2 -13016.593} C_VEL
LIN {X 0,Y 368.35,Z 163.559,A -85,B 0,C 180,E1 -13017.087,E2 -13017.087} C_VEL
LIN {X 0,Y 376.856,Z 180.701,A -85,B 0,C 180,E1 -13018.468,E2 -13018.468} C_VEL
LIN {X 0,Y 378.597,Z 184.897,A -85,B 0,C 180,E1 -13018.754,E2 -13018.754} C_VEL
LIN {X 0,Y 382.555,Z 205.182,A -85,B 0,C 180,E1 -13019.634,E2 -13019.634} C_VEL
LIN {X 0,Y 382.972,Z 209.268,A -85,B 0,C 180,E1 -13019.768,E2 -13019.768} C_VEL
LIN {X 0,Y 379.339,Z 330.828,A -85,B 0,C 180,E1 -13022.183,E2 -13022.183} C_VEL
LIN {X 0,Y 378.223,Z 346.43,A -85,B 0,C 180,E1 -13022.695,E2 -13022.695} C_VEL
LIN {X 0,Y 376.877,Z 360.234,A -85,B 0,C 180,E1 -13023.339,E2 -13023.339} C_VEL
LIN {X 0,Y 375.133,Z 375.245,A -85,B 0,C 180,E1 -13024.274,E2 -13024.274} C_VEL
LIN {X 0,Y 373.287,Z 389.083,A -85,B 0,C 180,E1 -13025.383,E2 -13025.383} C_VEL
LIN {X 0,Y 371.084,Z 402.571,A -85,B 0,C 180,E1 -13026.712,E2 -13026.712} C_VEL
LIN {X 0,Y 369.072,Z 414.848,A -85,B 0,C 180,E1 -13028.203,E2 -13028.203} C_VEL
LIN {X 0,Y 367.092,Z 426.07,A -85,B 0,C 180,E1 -13029.842,E2 -13029.842} C_VEL
LIN {X 0,Y 365.21,Z 437.028,A -85,B 0,C 180,E1 -13031.778,E2 -13031.778} C_VEL
LIN {X 0,Y 363.665,Z 446.133,A -85,B 0,C 180,E1 -13033.727,E2 -13033.727} C_VEL
LIN {X 0,Y 362.367,Z 453.796,A -85,B 0,C 180,E1 -13035.702,E2 -13035.702} C_VEL
LIN {X 0,Y 361.615,Z 460.051,A -85,B 0,C 180,E1 -13037.656,E2 -13037.656} C_VEL
LIN {X 0,Y 360.863,Z 465.888,A -85,B 0,C 180,E1 -13039.905,E2 -13039.905} C_VEL
LIN {X 0,Y 360.496,Z 470.392,A -85,B 0,C 180,E1 -13042.157,E2 -13042.157} C_VEL
LIN {X 0,Y 360.321,Z 473.649,A -85,B 0,C 180,E1 -13044.404,E2 -13044.404} C_VEL
LIN {X 0,Y 360.269,Z 475.666,A -85,B 0,C 180,E1 -13046.645,E2 -13046.645} C_VEL
LIN {X 0,Y 360.312,Z 476.534,A -85,B 0,C 180,E1 -13048.883,E2 -13048.883} C_VEL
LIN {X 0,Y 360.314,Z 476.263,A -85,B 0,C 180,E1 -13051.118,E2 -13051.118} C_VEL
LIN {X 0,Y 360.273,Z 474.838,A -85,B 0,C 180,E1 -13053.355,E2 -13053.355} C_VEL
LIN {X 0,Y 360.332,Z 472.216,A -85,B 0,C 180,E1 -13055.597,E2 -13055.597} C_VEL
LIN {X 0,Y 360.487,Z 468.302,A -85,B 0,C 180,E1 -13057.844,E2 -13057.844} C_VEL
LIN {X 0,Y 360.752,Z 463.036,A -85,B 0,C 180,E1 -13060.099,E2 -13060.099} C_VEL
LIN {X 0,Y 361.403,Z 456.292,A -85,B 0,C 180,E1 -13062.352,E2 -13062.352} C_VEL
LIN {X 0,Y 362.315,Z 447.868,A -85,B 0,C 180,E1 -13064.606,E2 -13064.606} C_VEL
LIN {X 0,Y 363.399,Z 438.853,A -85,B 0,C 180,E1 -13066.575,E2 -13066.575} C_VEL
LIN {X 0,Y 364.68,Z 429.66,A -85,B 0,C 180,E1 -13068.251,E2 -13068.251} C_VEL
LIN {X 0,Y 366.085,Z 418.973,A -85,B 0,C 180,E1 -13069.896,E2 -13069.896} C_VEL
LIN {X 0,Y 367.661,Z 406.904,A -85,B 0,C 180,E1 -13071.444,E2 -13071.444} C_VEL
LIN {X 0,Y 369.282,Z 393.908,A -85,B 0,C 180,E1 -13072.816,E2 -13072.816} C_VEL
LIN {X 0,Y 370.786,Z 381.349,A -85,B 0,C 180,E1 -13073.901,E2 -13073.901} C_VEL
LIN {X 0,Y 372.267,Z 367.031,A -85,B 0,C 180,E1 -13074.893,E2 -13074.893} C_VEL
LIN {X 0,Y 373.425,Z 352.199,A -85,B 0,C 180,E1 -13075.688,E2 -13075.688} C_VEL
LIN {X 0,Y 374.459,Z 337.568,A -85,B 0,C 180,E1 -13076.247,E2 -13076.247} C_VEL
LIN {X 0,Y 375.018,Z 321.303,A -85,B 0,C 180,E1 -13076.654,E2 -13076.654} C_VEL
LIN {X 0,Y 377.705,Z 206.38,A -85,B 0,C 180,E1 -13078.873,E2 -13078.873} C_VEL
LIN {X 0,Y 372.081,Z 175.678,A -85,B 0,C 180,E1 -13079.939,E2 -13079.939} C_VEL
LIN {X 0,Y 367.512,Z 164.145,A -85,B 0,C 180,E1 -13080.566,E2 -13080.566} C_VEL
LIN {X 0,Y 363.957,Z 149.111,A -85,B 0,C 180,E1 -13083.868,E2 -13083.868} C_VEL
